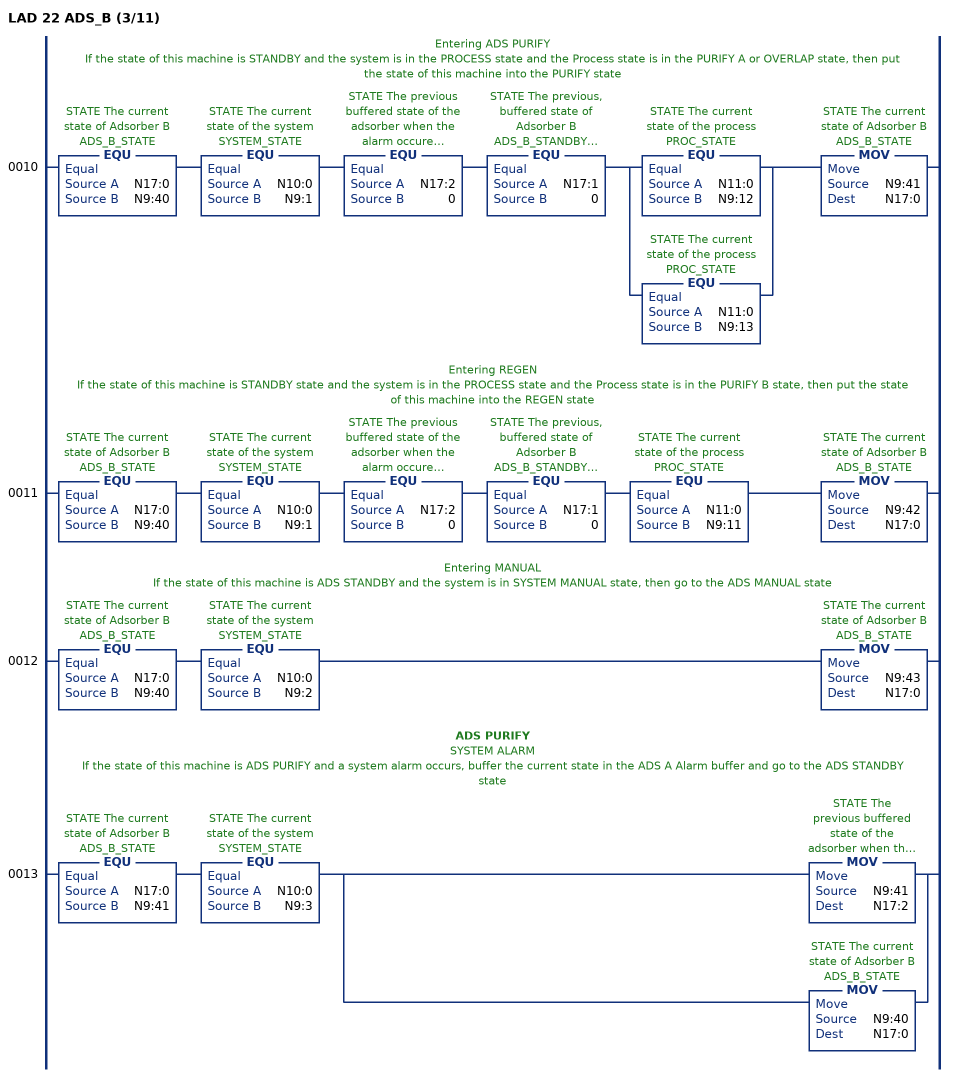
% Rung: 10 %
% Entering ADS PURIFY
% If the state of this machine is STANDBY and the system is in the PROCESS state and the Process state is in the PURIFY A or OVERLAP state, then put the state of this machine into the PURIFY state %
SOR EQU N17:0 N9:40 EQU N10:0 N9:1 EQU N17:2 0 EQU N17:1 0 BST EQU N11:0 N9:12 NXB EQU N11:0 N9:13 BND MOV N9:41 N17:0 EOR
%   N17:0  ADS_B_STATE  "STATE The current state of Adsorber B" %
%   N9:40  ADS_STANDBY  "STATE ADS Standby" %
%   N10:0  SYSTEM_STATE  "STATE The current state of the system" %
%   N9:1  SYSTEM_PROCESS  "STATE System Process" %
%   N17:2  ADS_B_SYS_ALARM_BUFR  "STATE The previous buffered state of the adsorber when the alarm occured" %
%   N17:1  ADS_B_STANDBY_BUFFER  "STATE The previous, buffered state of Adsorber B" %
%   N11:0  PROC_STATE  "STATE The current state of the process" %
%   N9:12  PROC_PURIFY_B  "STATE Process Purify B" %
%   N9:13  PROC_OVERLAP  "STATE Process Purify Overlap" %
%   N9:41  ADS_PURIFY  "STATE ADS Purify" %
% Rung: 11 %
% Entering REGEN
% If the state of this machine is STANDBY state and the system is in the PROCESS state and the Process state is in the PURIFY B state, then put the state of this machine into the REGEN state %
SOR EQU N17:0 N9:40 EQU N10:0 N9:1 EQU N17:2 0 EQU N17:1 0 EQU N11:0 N9:11 MOV N9:42 N17:0 EOR
%   N17:0  ADS_B_STATE  "STATE The current state of Adsorber B" %
%   N9:40  ADS_STANDBY  "STATE ADS Standby" %
%   N10:0  SYSTEM_STATE  "STATE The current state of the system" %
%   N9:1  SYSTEM_PROCESS  "STATE System Process" %
%   N17:2  ADS_B_SYS_ALARM_BUFR  "STATE The previous buffered state of the adsorber when the alarm occured" %
%   N17:1  ADS_B_STANDBY_BUFFER  "STATE The previous, buffered state of Adsorber B" %
%   N11:0  PROC_STATE  "STATE The current state of the process" %
%   N9:11  PROC_PURIFY_A  "STATE Process Purify A" %
%   N9:42  ADS_REGEN  "STATE ADS Regen" %
% Rung: 12 %
% Entering MANUAL
% If the state of this machine is ADS STANDBY and the system is in SYSTEM MANUAL state, then go to the ADS MANUAL state %
SOR EQU N17:0 N9:40 EQU N10:0 N9:2 MOV N9:43 N17:0 EOR
%   N17:0  ADS_B_STATE  "STATE The current state of Adsorber B" %
%   N9:40  ADS_STANDBY  "STATE ADS Standby" %
%   N10:0  SYSTEM_STATE  "STATE The current state of the system" %
%   N9:2  SYSTEM_MANUAL  "STATE System Manual" %
%   N9:43  ADS_MANUAL  "STATE ADS Manual" %
% Rung: 13 %
% TITLE: ADS PURIFY %
% SYSTEM ALARM
% If the state of this machine is ADS PURIFY and a system alarm occurs, buffer the current state in the ADS A Alarm buffer and go to the ADS STANDBY state %
SOR EQU N17:0 N9:41 EQU N10:0 N9:3 BST MOV N9:41 N17:2 NXB MOV N9:40 N17:0 BND EOR
%   N17:0  ADS_B_STATE  "STATE The current state of Adsorber B" %
%   N9:41  ADS_PURIFY  "STATE ADS Purify" %
%   N10:0  SYSTEM_STATE  "STATE The current state of the system" %
%   N9:3  SYSTEM_ALARM  "STATE System Alarm" %
%   N17:2  ADS_B_SYS_ALARM_BUFR  "STATE The previous buffered state of the adsorber when the alarm occured" %
%   N9:40  ADS_STANDBY  "STATE ADS Standby" %

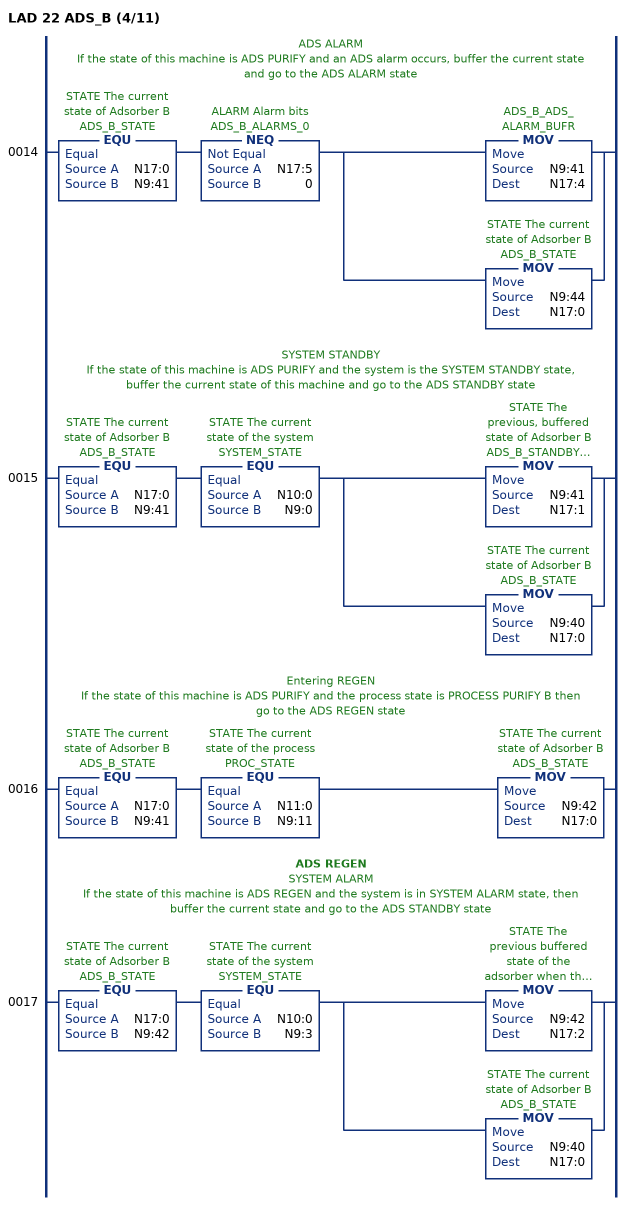
% Rung: 14 %
% ADS ALARM
% If the state of this machine is ADS PURIFY and an ADS alarm occurs, buffer the current state and go to the ADS ALARM state %
SOR EQU N17:0 N9:41 NEQ N17:5 0 BST MOV N9:41 N17:4 NXB MOV N9:44 N17:0 BND EOR
%   N17:0  ADS_B_STATE  "STATE The current state of Adsorber B" %
%   N9:41  ADS_PURIFY  "STATE ADS Purify" %
%   N17:5  ADS_B_ALARMS_0  "ALARM Alarm bits" %
%   N17:4  ADS_B_ADS_ALARM_BUFR %
%   N9:44  ADS_ALARM  "STATE ADS Alarm" %
% Rung: 15 %
% SYSTEM STANDBY
% If the state of this machine is ADS PURIFY and the system is the SYSTEM STANDBY state, buffer the current state of this machine and go to the ADS STANDBY state %
SOR EQU N17:0 N9:41 EQU N10:0 N9:0 BST MOV N9:41 N17:1 NXB MOV N9:40 N17:0 BND EOR
%   N17:0  ADS_B_STATE  "STATE The current state of Adsorber B" %
%   N9:41  ADS_PURIFY  "STATE ADS Purify" %
%   N10:0  SYSTEM_STATE  "STATE The current state of the system" %
%   N9:0  SYSTEM_STANDBY  "STATE System Standby" %
%   N17:1  ADS_B_STANDBY_BUFFER  "STATE The previous, buffered state of Adsorber B" %
%   N9:40  ADS_STANDBY  "STATE ADS Standby" %
% Rung: 16 %
% Entering REGEN
% If the state of this machine is ADS PURIFY and the process state is PROCESS PURIFY B then go to the ADS REGEN state %
SOR EQU N17:0 N9:41 EQU N11:0 N9:11 MOV N9:42 N17:0 EOR
%   N17:0  ADS_B_STATE  "STATE The current state of Adsorber B" %
%   N9:41  ADS_PURIFY  "STATE ADS Purify" %
%   N11:0  PROC_STATE  "STATE The current state of the process" %
%   N9:11  PROC_PURIFY_A  "STATE Process Purify A" %
%   N9:42  ADS_REGEN  "STATE ADS Regen" %
% Rung: 17 %
% TITLE: ADS REGEN %
% SYSTEM ALARM
% If the state of this machine is ADS REGEN and the system is in SYSTEM ALARM state, then buffer the current state and go to the ADS STANDBY state %
SOR EQU N17:0 N9:42 EQU N10:0 N9:3 BST MOV N9:42 N17:2 NXB MOV N9:40 N17:0 BND EOR
%   N17:0  ADS_B_STATE  "STATE The current state of Adsorber B" %
%   N9:42  ADS_REGEN  "STATE ADS Regen" %
%   N10:0  SYSTEM_STATE  "STATE The current state of the system" %
%   N9:3  SYSTEM_ALARM  "STATE System Alarm" %
%   N17:2  ADS_B_SYS_ALARM_BUFR  "STATE The previous buffered state of the adsorber when the alarm occured" %
%   N9:40  ADS_STANDBY  "STATE ADS Standby" %

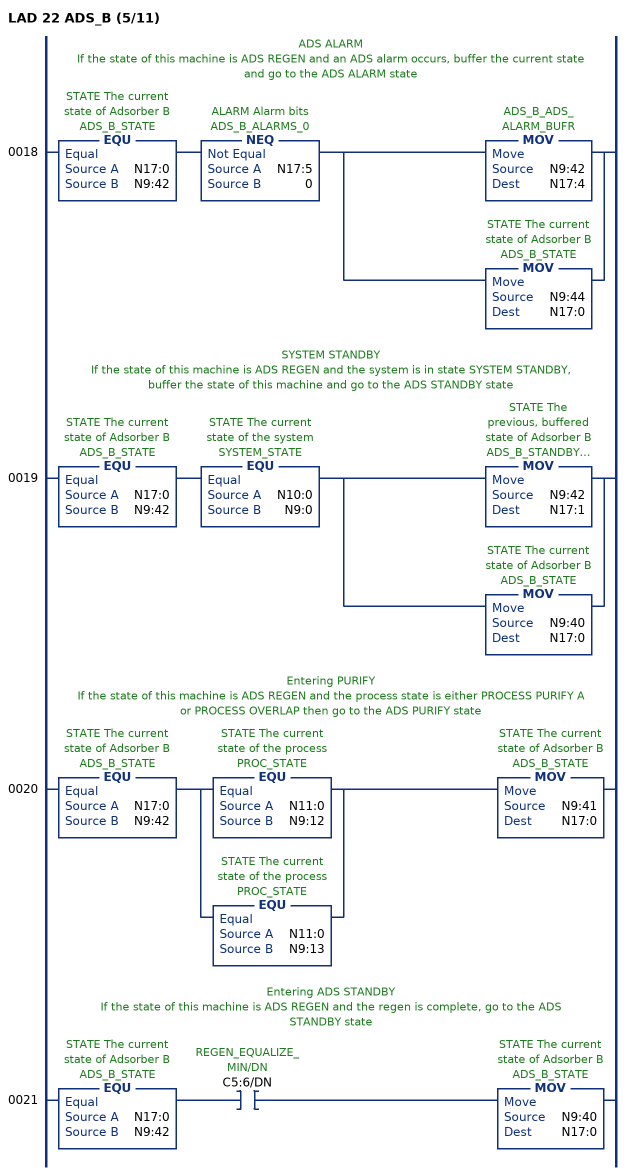
% Rung: 18 %
% ADS ALARM
% If the state of this machine is ADS REGEN and an ADS alarm occurs, buffer the current state and go to the ADS ALARM state %
SOR EQU N17:0 N9:42 NEQ N17:5 0 BST MOV N9:42 N17:4 NXB MOV N9:44 N17:0 BND EOR
%   N17:0  ADS_B_STATE  "STATE The current state of Adsorber B" %
%   N9:42  ADS_REGEN  "STATE ADS Regen" %
%   N17:5  ADS_B_ALARMS_0  "ALARM Alarm bits" %
%   N17:4  ADS_B_ADS_ALARM_BUFR %
%   N9:44  ADS_ALARM  "STATE ADS Alarm" %
% Rung: 19 %
% SYSTEM STANDBY
% If the state of this machine is ADS REGEN and the system is in state SYSTEM STANDBY, buffer the state of this machine and go to the ADS STANDBY state %
SOR EQU N17:0 N9:42 EQU N10:0 N9:0 BST MOV N9:42 N17:1 NXB MOV N9:40 N17:0 BND EOR
%   N17:0  ADS_B_STATE  "STATE The current state of Adsorber B" %
%   N9:42  ADS_REGEN  "STATE ADS Regen" %
%   N10:0  SYSTEM_STATE  "STATE The current state of the system" %
%   N9:0  SYSTEM_STANDBY  "STATE System Standby" %
%   N17:1  ADS_B_STANDBY_BUFFER  "STATE The previous, buffered state of Adsorber B" %
%   N9:40  ADS_STANDBY  "STATE ADS Standby" %
% Rung: 20 %
% Entering PURIFY
% If the state of this machine is ADS REGEN and the process state is either PROCESS PURIFY A or PROCESS OVERLAP then go to the ADS PURIFY state %
SOR EQU N17:0 N9:42 BST EQU N11:0 N9:12 NXB EQU N11:0 N9:13 BND MOV N9:41 N17:0 EOR
%   N17:0  ADS_B_STATE  "STATE The current state of Adsorber B" %
%   N9:42  ADS_REGEN  "STATE ADS Regen" %
%   N11:0  PROC_STATE  "STATE The current state of the process" %
%   N9:12  PROC_PURIFY_B  "STATE Process Purify B" %
%   N9:13  PROC_OVERLAP  "STATE Process Purify Overlap" %
%   N9:41  ADS_PURIFY  "STATE ADS Purify" %
% Rung: 21 %
% Entering ADS STANDBY
% If the state of this machine is ADS REGEN and the regen is complete, go to the ADS STANDBY state %
SOR EQU N17:0 N9:42 XIC C5:6/DN MOV N9:40 N17:0 EOR
%   N17:0  ADS_B_STATE  "STATE The current state of Adsorber B" %
%   N9:42  ADS_REGEN  "STATE ADS Regen" %
%   C5:6  REGEN_EQUALIZE_MIN %
%   N9:40  ADS_STANDBY  "STATE ADS Standby" %

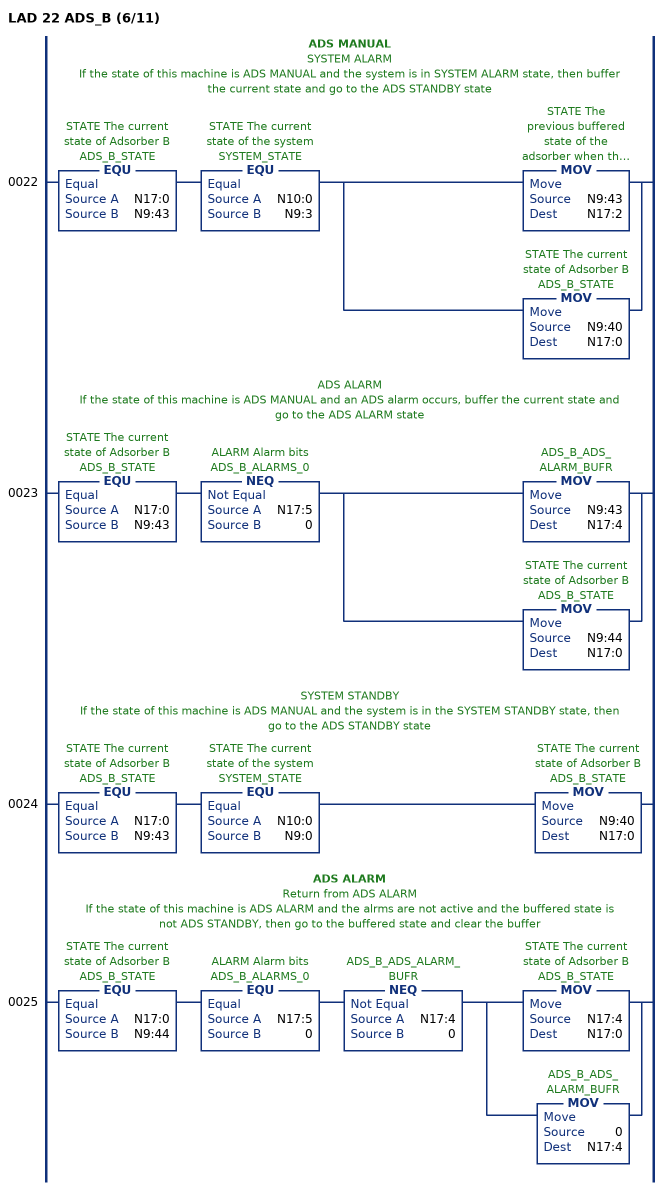
% Rung: 22 %
% TITLE: ADS MANUAL %
% SYSTEM ALARM
% If the state of this machine is ADS MANUAL and the system is in SYSTEM ALARM state, then buffer the current state and go to the ADS STANDBY state %
SOR EQU N17:0 N9:43 EQU N10:0 N9:3 BST MOV N9:43 N17:2 NXB MOV N9:40 N17:0 BND EOR
%   N17:0  ADS_B_STATE  "STATE The current state of Adsorber B" %
%   N9:43  ADS_MANUAL  "STATE ADS Manual" %
%   N10:0  SYSTEM_STATE  "STATE The current state of the system" %
%   N9:3  SYSTEM_ALARM  "STATE System Alarm" %
%   N17:2  ADS_B_SYS_ALARM_BUFR  "STATE The previous buffered state of the adsorber when the alarm occured" %
%   N9:40  ADS_STANDBY  "STATE ADS Standby" %
% Rung: 23 %
% ADS ALARM
% If the state of this machine is ADS MANUAL and an ADS alarm occurs, buffer the current state and go to the ADS ALARM state %
SOR EQU N17:0 N9:43 NEQ N17:5 0 BST MOV N9:43 N17:4 NXB MOV N9:44 N17:0 BND EOR
%   N17:0  ADS_B_STATE  "STATE The current state of Adsorber B" %
%   N9:43  ADS_MANUAL  "STATE ADS Manual" %
%   N17:5  ADS_B_ALARMS_0  "ALARM Alarm bits" %
%   N17:4  ADS_B_ADS_ALARM_BUFR %
%   N9:44  ADS_ALARM  "STATE ADS Alarm" %
% Rung: 24 %
% SYSTEM STANDBY
% If the state of this machine is ADS MANUAL and the system is in the SYSTEM STANDBY state, then go to the ADS STANDBY state %
SOR EQU N17:0 N9:43 EQU N10:0 N9:0 MOV N9:40 N17:0 EOR
%   N17:0  ADS_B_STATE  "STATE The current state of Adsorber B" %
%   N9:43  ADS_MANUAL  "STATE ADS Manual" %
%   N10:0  SYSTEM_STATE  "STATE The current state of the system" %
%   N9:0  SYSTEM_STANDBY  "STATE System Standby" %
%   N9:40  ADS_STANDBY  "STATE ADS Standby" %
% Rung: 25 %
% TITLE: ADS ALARM %
% Return from ADS ALARM
% If the state of this machine is ADS ALARM and the alrms are not active and the buffered state is not ADS STANDBY, then go to the buffered state and clear the buffer %
SOR EQU N17:0 N9:44 EQU N17:5 0 NEQ N17:4 0 BST MOV N17:4 N17:0 NXB MOV 0 N17:4 BND EOR
%   N17:0  ADS_B_STATE  "STATE The current state of Adsorber B" %
%   N9:44  ADS_ALARM  "STATE ADS Alarm" %
%   N17:5  ADS_B_ALARMS_0  "ALARM Alarm bits" %
%   N17:4  ADS_B_ADS_ALARM_BUFR %

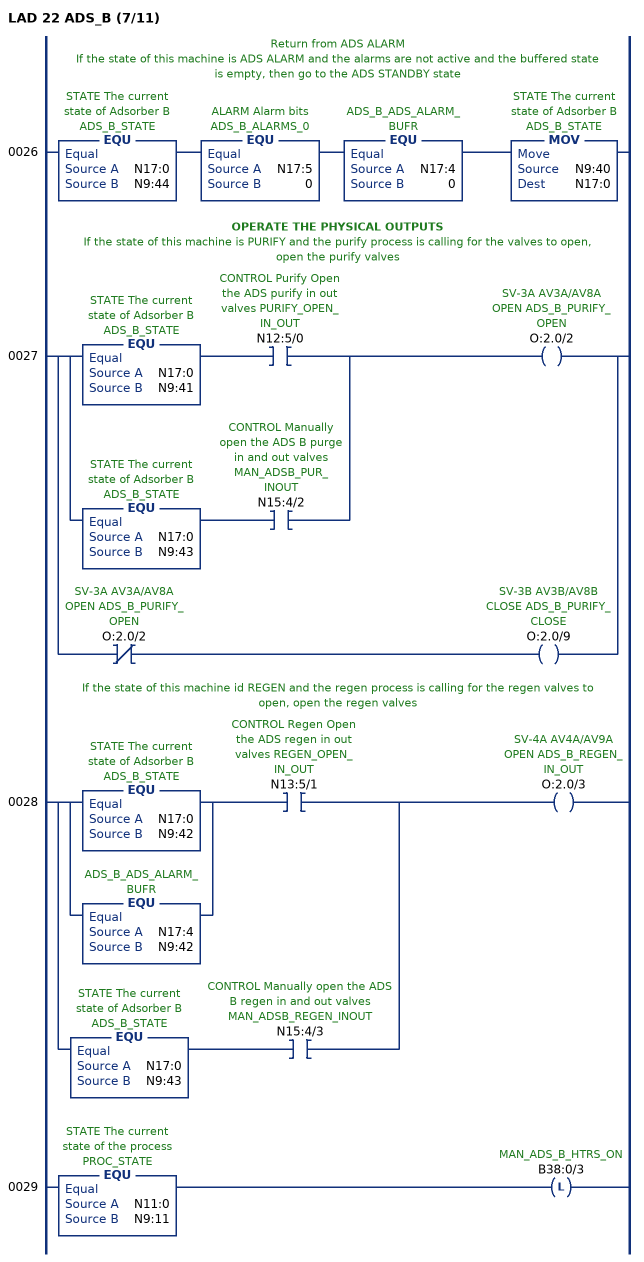
% Rung: 26 %
% Return from ADS ALARM
% If the state of this machine is ADS ALARM and the alarms are not active and the buffered state is empty, then go to the ADS STANDBY state %
SOR EQU N17:0 N9:44 EQU N17:5 0 EQU N17:4 0 MOV N9:40 N17:0 EOR
%   N17:0  ADS_B_STATE  "STATE The current state of Adsorber B" %
%   N9:44  ADS_ALARM  "STATE ADS Alarm" %
%   N17:5  ADS_B_ALARMS_0  "ALARM Alarm bits" %
%   N17:4  ADS_B_ADS_ALARM_BUFR %
%   N9:40  ADS_STANDBY  "STATE ADS Standby" %
% Rung: 27 %
% TITLE: OPERATE THE PHYSICAL OUTPUTS %
% If the state of this machine is PURIFY and the purify process is calling for the valves to open, open the purify valves %
SOR BST BST EQU N17:0 N9:41 XIC N12:5/0 NXB EQU N17:0 N9:43 XIC N15:4/2 BND OTE O:2.0/2 NXB XIO O:2.0/2 OTE O:2.0/9 BND EOR
%   N17:0  ADS_B_STATE  "STATE The current state of Adsorber B" %
%   N9:41  ADS_PURIFY  "STATE ADS Purify" %
%   N12:5/0  PURIFY_OPEN_IN_OUT  "CONTROL Purify Open the ADS purify in out valves" %
%   N9:43  ADS_MANUAL  "STATE ADS Manual" %
%   N15:4/2  MAN_ADSB_PUR_INOUT  "CONTROL Manually open the ADS B purge in and out valves" %
%   O:2.0/2  ADS_B_PURIFY_OPEN  "SV-3A AV3A/AV8A OPEN" %
%   O:2.0/9  ADS_B_PURIFY_CLOSE  "SV-3B AV3B/AV8B CLOSE" %
% Rung: 28 %
% If the state of this machine id REGEN and the regen process is calling for the regen valves to open, open the regen valves %
SOR BST BST EQU N17:0 N9:42 NXB EQU N17:4 N9:42 BND XIC N13:5/1 NXB EQU N17:0 N9:43 XIC N15:4/3 BND OTE O:2.0/3 EOR
%   N17:0  ADS_B_STATE  "STATE The current state of Adsorber B" %
%   N9:42  ADS_REGEN  "STATE ADS Regen" %
%   N17:4  ADS_B_ADS_ALARM_BUFR %
%   N13:5/1  REGEN_OPEN_IN_OUT  "CONTROL Regen Open the ADS regen in out valves" %
%   N9:43  ADS_MANUAL  "STATE ADS Manual" %
%   N15:4/3  MAN_ADSB_REGEN_INOUT  "CONTROL Manually open the ADS B regen in and out valves" %
%   O:2.0/3  ADS_B_REGEN_IN_OUT  "SV-4A AV4A/AV9A OPEN" %
% Rung: 29 %
SOR EQU N11:0 N9:11 OTL B38:0/3 EOR
%   N11:0  PROC_STATE  "STATE The current state of the process" %
%   N9:11  PROC_PURIFY_A  "STATE Process Purify A" %
%   B38:0/3  MAN_ADS_B_HTRS_ON %

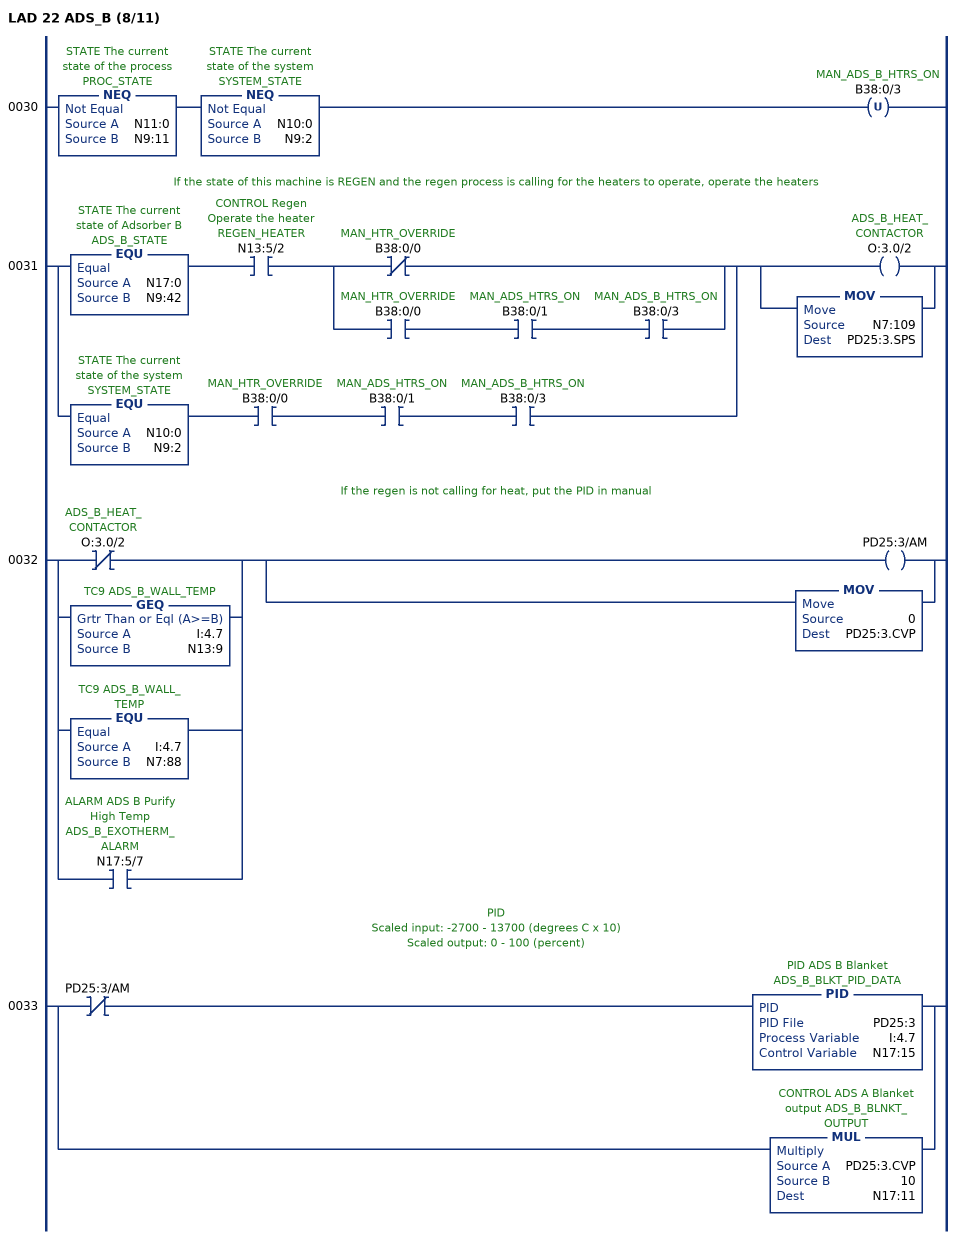
% Rung: 30 %
SOR NEQ N11:0 N9:11 NEQ N10:0 N9:2 OTU B38:0/3 EOR
%   N11:0  PROC_STATE  "STATE The current state of the process" %
%   N9:11  PROC_PURIFY_A  "STATE Process Purify A" %
%   N10:0  SYSTEM_STATE  "STATE The current state of the system" %
%   N9:2  SYSTEM_MANUAL  "STATE System Manual" %
%   B38:0/3  MAN_ADS_B_HTRS_ON %
% Rung: 31 %
% If the state of this machine is REGEN and the regen process is calling for the heaters to operate, operate the heaters %
SOR BST EQU N17:0 N9:42 XIC N13:5/2 BST XIO B38:0/0 NXB XIC B38:0/0 XIC B38:0/1 XIC B38:0/3 BND NXB EQU N10:0 N9:2 XIC B38:0/0 XIC B38:0/1 XIC B38:0/3 BND BST OTE O:3.0/2 NXB MOV N7:109 PD25:3.SPS BND EOR
%   N17:0  ADS_B_STATE  "STATE The current state of Adsorber B" %
%   N9:42  ADS_REGEN  "STATE ADS Regen" %
%   N13:5/2  REGEN_HEATER  "CONTROL Regen Operate the heater" %
%   B38:0/0  MAN_HTR_OVERRIDE %
%   B38:0/1  MAN_ADS_HTRS_ON %
%   B38:0/3  MAN_ADS_B_HTRS_ON %
%   N10:0  SYSTEM_STATE  "STATE The current state of the system" %
%   N9:2  SYSTEM_MANUAL  "STATE System Manual" %
%   O:3.0/2  ADS_B_HEAT_CONTACTOR %
%   N7:109  BLANKET_SP  "CONTROL Blanket PID Setpoint" %
% Rung: 32 %
% If the regen is not calling for heat, put the PID in manual %
SOR BST XIO O:3.0/2 NXB GEQ I:4.7 N13:9 NXB EQU I:4.7 N7:88 NXB XIC N17:5/7 BND BST OTE PD25:3/AM NXB MOV 0 PD25:3.CVP BND EOR
%   O:3.0/2  ADS_B_HEAT_CONTACTOR %
%   I:4.7  ADS_B_WALL_TEMP  "TC9" %
%   N13:9  BLANKET_LIMIT %
%   N7:88  TC_OPEN_SP  "CONFIG The value read by an open TC input" %
%   N17:5/7  ADS_B_EXOTHERM_ALARM  "ALARM ADS B Purify High Temp" %
% Rung: 33 %
% PID
% Scaled input: -2700 - 13700 (degrees C x 10)
% Scaled output: 0 - 100 (percent) %
SOR BST XIO PD25:3/AM PID PD25:3 I:4.7 N17:15 NXB MUL PD25:3.CVP 10 N17:11 BND EOR
%   PD25:3  ADS_B_BLKT_PID_DATA  "PID ADS B Blanket" %
%   I:4.7  ADS_B_WALL_TEMP  "TC9" %
%   N17:15  ADS_B_BLKT_OUTPT_RAW  "CONTROL ADS B Blanket PID Output Raw" %
%   N17:11  ADS_B_BLNKT_OUTPUT  "CONTROL ADS A Blanket output" %

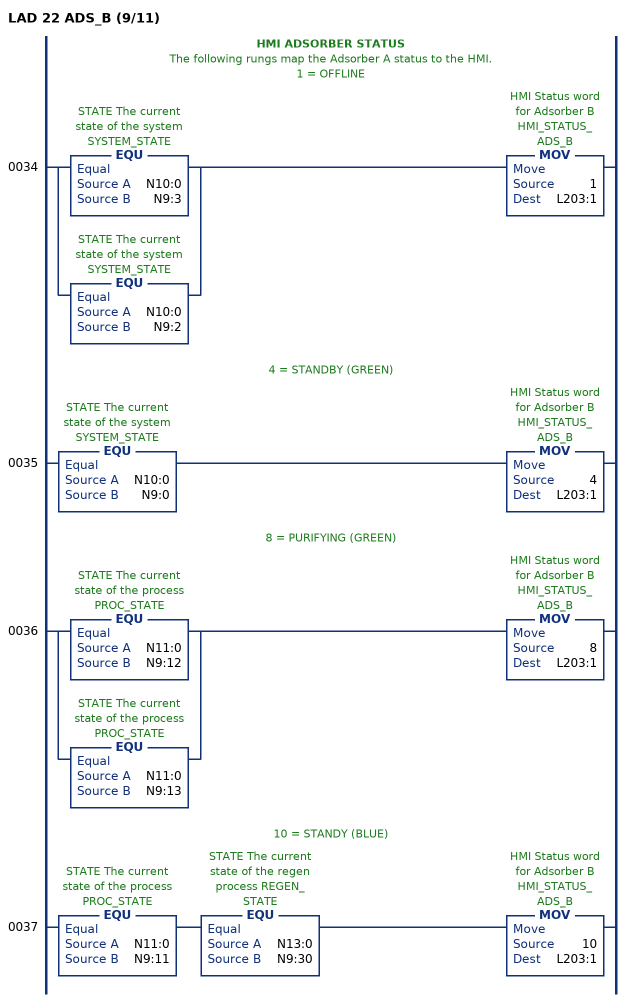
% Rung: 34 %
% TITLE: HMI ADSORBER STATUS %
% The following rungs map the Adsorber A status to the HMI.
% 1 = OFFLINE %
SOR BST EQU N10:0 N9:3 NXB EQU N10:0 N9:2 BND MOV 1 L203:1 EOR
%   N10:0  SYSTEM_STATE  "STATE The current state of the system" %
%   N9:3  SYSTEM_ALARM  "STATE System Alarm" %
%   N9:2  SYSTEM_MANUAL  "STATE System Manual" %
%   L203:1  HMI_STATUS_ADS_B  "HMI Status word for Adsorber B" %
% Rung: 35 %
% 4 = STANDBY (GREEN) %
SOR EQU N10:0 N9:0 MOV 4 L203:1 EOR
%   N10:0  SYSTEM_STATE  "STATE The current state of the system" %
%   N9:0  SYSTEM_STANDBY  "STATE System Standby" %
%   L203:1  HMI_STATUS_ADS_B  "HMI Status word for Adsorber B" %
% Rung: 36 %
% 8 = PURIFYING (GREEN) %
SOR BST EQU N11:0 N9:12 NXB EQU N11:0 N9:13 BND MOV 8 L203:1 EOR
%   N11:0  PROC_STATE  "STATE The current state of the process" %
%   N9:12  PROC_PURIFY_B  "STATE Process Purify B" %
%   N9:13  PROC_OVERLAP  "STATE Process Purify Overlap" %
%   L203:1  HMI_STATUS_ADS_B  "HMI Status word for Adsorber B" %
% Rung: 37 %
% 10 = STANDY (BLUE) %
SOR EQU N11:0 N9:11 EQU N13:0 N9:30 MOV 10 L203:1 EOR
%   N11:0  PROC_STATE  "STATE The current state of the process" %
%   N9:11  PROC_PURIFY_A  "STATE Process Purify A" %
%   N13:0  REGEN_STATE  "STATE The current state of the regen process" %
%   N9:30  REGEN_STANDBY  "STATE Regen Standby" %
%   L203:1  HMI_STATUS_ADS_B  "HMI Status word for Adsorber B" %

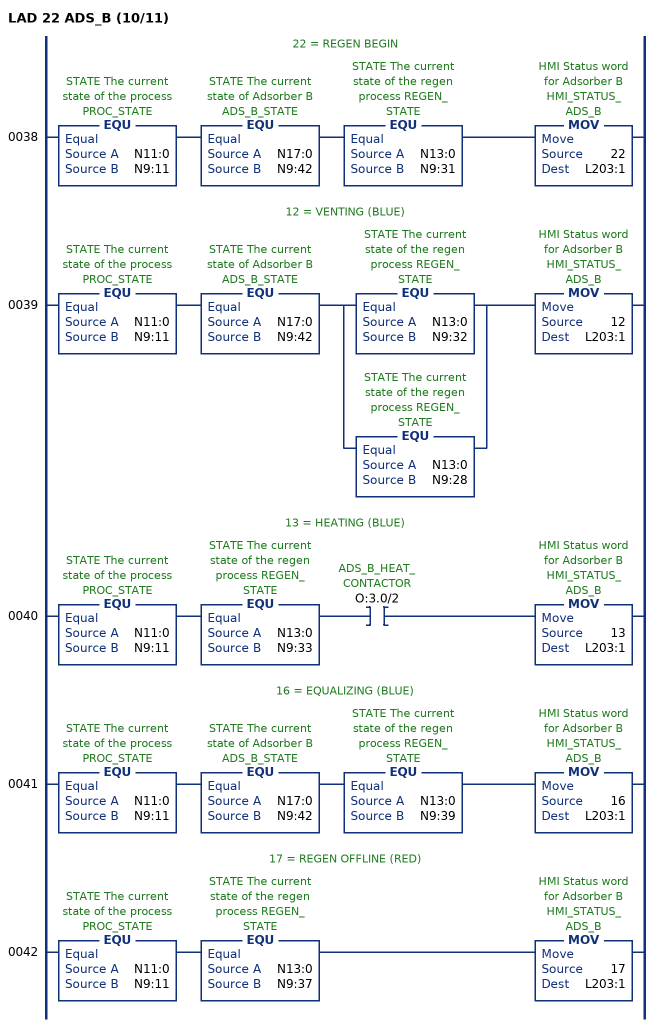
% Rung: 38 %
% 22 = REGEN BEGIN %
SOR EQU N11:0 N9:11 EQU N17:0 N9:42 EQU N13:0 N9:31 MOV 22 L203:1 EOR
%   N11:0  PROC_STATE  "STATE The current state of the process" %
%   N9:11  PROC_PURIFY_A  "STATE Process Purify A" %
%   N17:0  ADS_B_STATE  "STATE The current state of Adsorber B" %
%   N9:42  ADS_REGEN  "STATE ADS Regen" %
%   N13:0  REGEN_STATE  "STATE The current state of the regen process" %
%   N9:31  REGEN_DELAY  "STATE Regen Delay" %
%   L203:1  HMI_STATUS_ADS_B  "HMI Status word for Adsorber B" %
% Rung: 39 %
% 12 = VENTING (BLUE) %
SOR EQU N11:0 N9:11 EQU N17:0 N9:42 BST EQU N13:0 N9:32 NXB EQU N13:0 N9:28 BND MOV 12 L203:1 EOR
%   N11:0  PROC_STATE  "STATE The current state of the process" %
%   N9:11  PROC_PURIFY_A  "STATE Process Purify A" %
%   N17:0  ADS_B_STATE  "STATE The current state of Adsorber B" %
%   N9:42  ADS_REGEN  "STATE ADS Regen" %
%   N13:0  REGEN_STATE  "STATE The current state of the regen process" %
%   N9:32  REGEN_VENT  "STATE Regen Vent" %
%   N9:28  REGEN_VENT_2  "STATE Regen Vent 2" %
%   L203:1  HMI_STATUS_ADS_B  "HMI Status word for Adsorber B" %
% Rung: 40 %
% 13 = HEATING (BLUE) %
SOR EQU N11:0 N9:11 EQU N13:0 N9:33 XIC O:3.0/2 MOV 13 L203:1 EOR
%   N11:0  PROC_STATE  "STATE The current state of the process" %
%   N9:11  PROC_PURIFY_A  "STATE Process Purify A" %
%   N13:0  REGEN_STATE  "STATE The current state of the regen process" %
%   N9:33  REGEN_HEAT_BED  "STATE Regen Heat wall" %
%   O:3.0/2  ADS_B_HEAT_CONTACTOR %
%   L203:1  HMI_STATUS_ADS_B  "HMI Status word for Adsorber B" %
% Rung: 41 %
% 16 = EQUALIZING (BLUE) %
SOR EQU N11:0 N9:11 EQU N17:0 N9:42 EQU N13:0 N9:39 MOV 16 L203:1 EOR
%   N11:0  PROC_STATE  "STATE The current state of the process" %
%   N9:11  PROC_PURIFY_A  "STATE Process Purify A" %
%   N17:0  ADS_B_STATE  "STATE The current state of Adsorber B" %
%   N9:42  ADS_REGEN  "STATE ADS Regen" %
%   N13:0  REGEN_STATE  "STATE The current state of the regen process" %
%   N9:39  REGEN_EQUALIZE %
%   L203:1  HMI_STATUS_ADS_B  "HMI Status word for Adsorber B" %
% Rung: 42 %
% 17 = REGEN OFFLINE (RED) %
SOR EQU N11:0 N9:11 EQU N13:0 N9:37 MOV 17 L203:1 EOR
%   N11:0  PROC_STATE  "STATE The current state of the process" %
%   N9:11  PROC_PURIFY_A  "STATE Process Purify A" %
%   N13:0  REGEN_STATE  "STATE The current state of the regen process" %
%   N9:37  REGEN_ALARM  "STATE Regen Alarm" %
%   L203:1  HMI_STATUS_ADS_B  "HMI Status word for Adsorber B" %

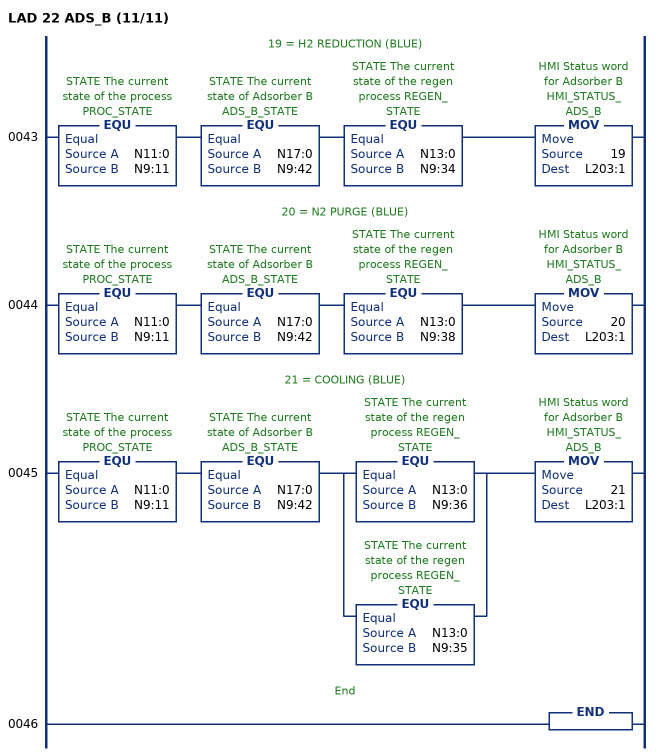
% Rung: 43 %
% 19 = H2 REDUCTION (BLUE) %
SOR EQU N11:0 N9:11 EQU N17:0 N9:42 EQU N13:0 N9:34 MOV 19 L203:1 EOR
%   N11:0  PROC_STATE  "STATE The current state of the process" %
%   N9:11  PROC_PURIFY_A  "STATE Process Purify A" %
%   N17:0  ADS_B_STATE  "STATE The current state of Adsorber B" %
%   N9:42  ADS_REGEN  "STATE ADS Regen" %
%   N13:0  REGEN_STATE  "STATE The current state of the regen process" %
%   N9:34  REGEN_H2_REDUCTION  "STATE Regen Running" %
%   L203:1  HMI_STATUS_ADS_B  "HMI Status word for Adsorber B" %
% Rung: 44 %
% 20 = N2 PURGE (BLUE) %
SOR EQU N11:0 N9:11 EQU N17:0 N9:42 EQU N13:0 N9:38 MOV 20 L203:1 EOR
%   N11:0  PROC_STATE  "STATE The current state of the process" %
%   N9:11  PROC_PURIFY_A  "STATE Process Purify A" %
%   N17:0  ADS_B_STATE  "STATE The current state of Adsorber B" %
%   N9:42  ADS_REGEN  "STATE ADS Regen" %
%   N13:0  REGEN_STATE  "STATE The current state of the regen process" %
%   N9:38  REGEN_PURGE  "STATE Regen Hot Purge" %
%   L203:1  HMI_STATUS_ADS_B  "HMI Status word for Adsorber B" %
% Rung: 45 %
% 21 = COOLING (BLUE) %
SOR EQU N11:0 N9:11 EQU N17:0 N9:42 BST EQU N13:0 N9:36 NXB EQU N13:0 N9:35 BND MOV 21 L203:1 EOR
%   N11:0  PROC_STATE  "STATE The current state of the process" %
%   N9:11  PROC_PURIFY_A  "STATE Process Purify A" %
%   N17:0  ADS_B_STATE  "STATE The current state of Adsorber B" %
%   N9:42  ADS_REGEN  "STATE ADS Regen" %
%   N13:0  REGEN_STATE  "STATE The current state of the regen process" %
%   N9:36  REGEN_COOL  "STATE Regen Cool" %
%   N9:35  REGEN_COOL_WALL  "STATE Regen Cool wall" %
%   L203:1  HMI_STATUS_ADS_B  "HMI Status word for Adsorber B" %
% Rung: 46 %
% End %
SOR END EOR

LADDER 23 "ADS_B_FLT"    % Controls the Adsorber B faults %
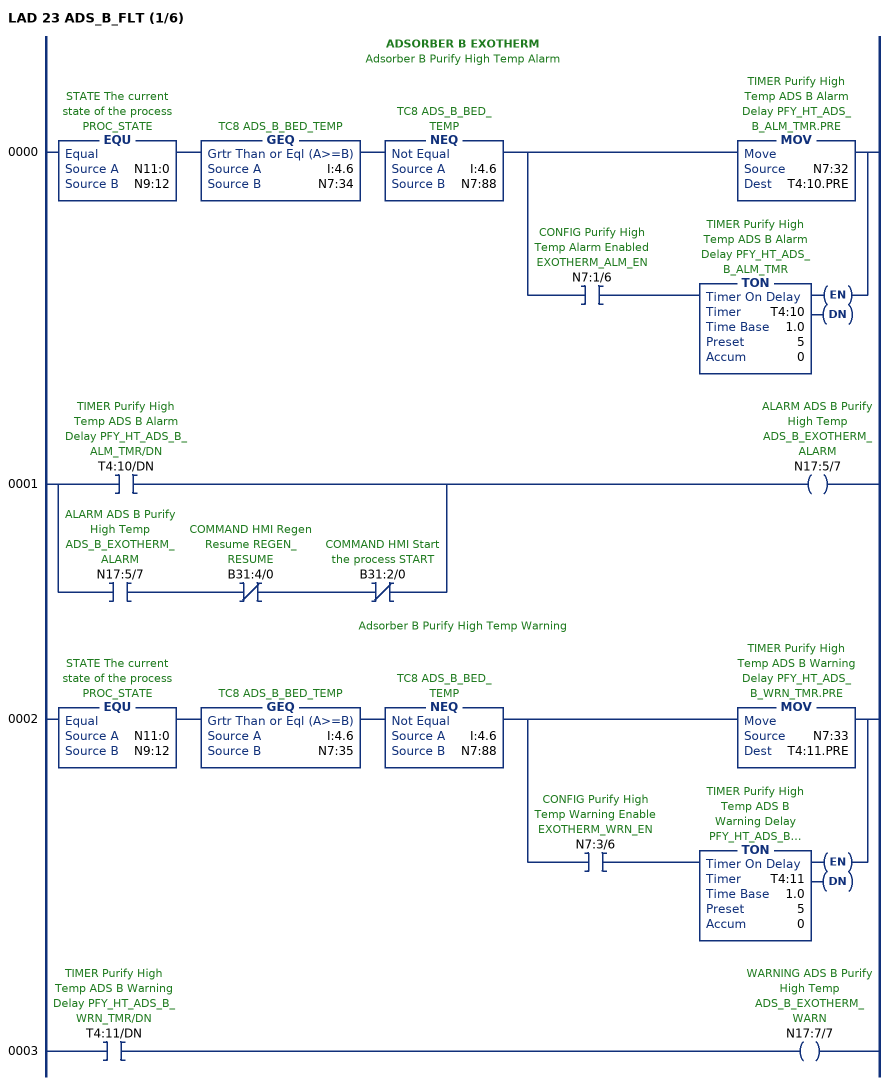
% Rung: 0 %
% TITLE: ADSORBER B EXOTHERM %
% Adsorber B Purify High Temp Alarm %
SOR EQU N11:0 N9:12 GEQ I:4.6 N7:34 NEQ I:4.6 N7:88 BST MOV N7:32 T4:10.PRE NXB XIC N7:1/6 TON T4:10 1.0 5 0 BND EOR
%   N11:0  PROC_STATE  "STATE The current state of the process" %
%   N9:12  PROC_PURIFY_B  "STATE Process Purify B" %
%   I:4.6  ADS_B_BED_TEMP  "TC8" %
%   N7:34  EXOTHERM_ALM_SP  "CONFIG Purify High Temp Alarm Setpoint" %
%   N7:88  TC_OPEN_SP  "CONFIG The value read by an open TC input" %
%   N7:32  EXOTHERM_ALM_DLY  "CONFIG Purify High Temp Alarm Delay" %
%   T4:10  PFY_HT_ADS_B_ALM_TMR  "TIMER Purify High Temp ADS B Alarm Delay" %
%   N7:1/6  EXOTHERM_ALM_EN  "CONFIG Purify High Temp Alarm Enabled" %
% Rung: 1 %
SOR BST XIC T4:10/DN NXB XIC N17:5/7 XIO B31:4/0 XIO B31:2/0 BND OTE N17:5/7 EOR
%   T4:10  PFY_HT_ADS_B_ALM_TMR  "TIMER Purify High Temp ADS B Alarm Delay" %
%   N17:5/7  ADS_B_EXOTHERM_ALARM  "ALARM ADS B Purify High Temp" %
%   B31:4/0  REGEN_RESUME  "COMMAND HMI Regen Resume" %
%   B31:2/0  START  "COMMAND HMI Start the process" %
% Rung: 2 %
% Adsorber B Purify High Temp Warning %
SOR EQU N11:0 N9:12 GEQ I:4.6 N7:35 NEQ I:4.6 N7:88 BST MOV N7:33 T4:11.PRE NXB XIC N7:3/6 TON T4:11 1.0 5 0 BND EOR
%   N11:0  PROC_STATE  "STATE The current state of the process" %
%   N9:12  PROC_PURIFY_B  "STATE Process Purify B" %
%   I:4.6  ADS_B_BED_TEMP  "TC8" %
%   N7:35  EXOTHERM_WRN_SP  "CONFIG Purify High Temp Warning Setpoint" %
%   N7:88  TC_OPEN_SP  "CONFIG The value read by an open TC input" %
%   N7:33  EXOTHERM_WRN_DLY  "CONFIG Purify High Temp Warning Delay" %
%   T4:11  PFY_HT_ADS_B_WRN_TMR  "TIMER Purify High Temp ADS B Warning Delay" %
%   N7:3/6  EXOTHERM_WRN_EN  "CONFIG Purify High Temp Warning Enable" %
% Rung: 3 %
SOR XIC T4:11/DN OTE N17:7/7 EOR
%   T4:11  PFY_HT_ADS_B_WRN_TMR  "TIMER Purify High Temp ADS B Warning Delay" %
%   N17:7/7  ADS_B_EXOTHERM_WARN  "WARNING ADS B Purify High Temp" %

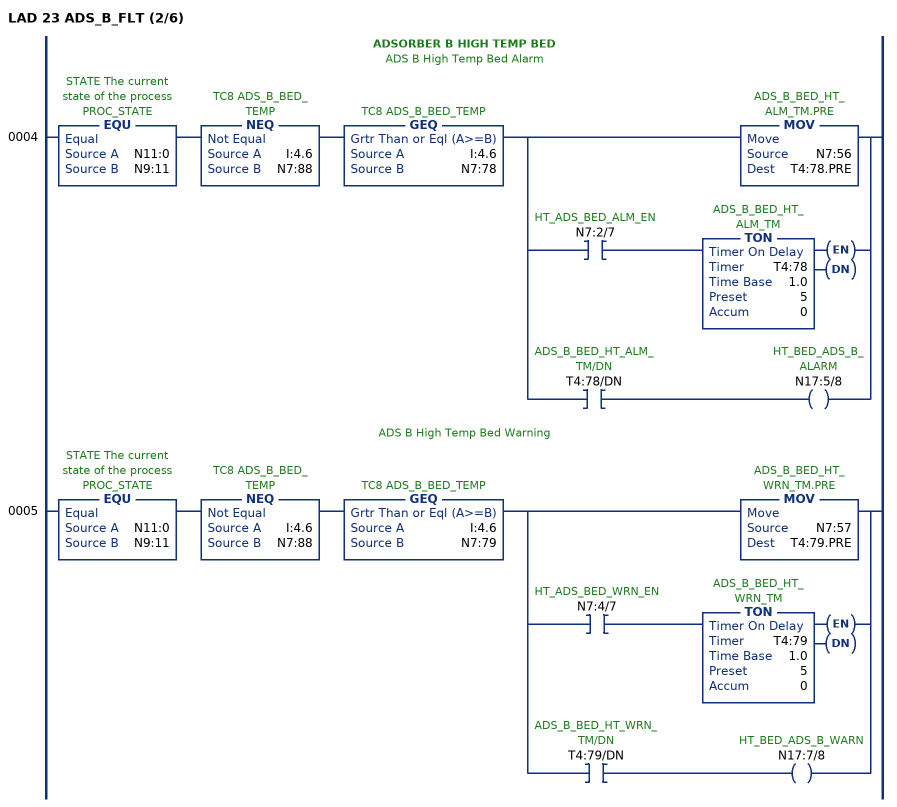
% Rung: 4 %
% TITLE: ADSORBER B HIGH TEMP BED %
% ADS B High Temp Bed Alarm %
SOR EQU N11:0 N9:11 NEQ I:4.6 N7:88 GEQ I:4.6 N7:78 BST MOV N7:56 T4:78.PRE NXB XIC N7:2/7 TON T4:78 1.0 5 0 NXB XIC T4:78/DN OTE N17:5/8 BND EOR
%   N11:0  PROC_STATE  "STATE The current state of the process" %
%   N9:11  PROC_PURIFY_A  "STATE Process Purify A" %
%   I:4.6  ADS_B_BED_TEMP  "TC8" %
%   N7:88  TC_OPEN_SP  "CONFIG The value read by an open TC input" %
%   N7:78  HT_ADS_BED_ALM_SP %
%   N7:56  HT_ADS_BED_ALM_DLY %
%   T4:78  ADS_B_BED_HT_ALM_TM %
%   N7:2/7  HT_ADS_BED_ALM_EN %
%   N17:5/8  HT_BED_ADS_B_ALARM %
% Rung: 5 %
% ADS B High Temp Bed Warning %
SOR EQU N11:0 N9:11 NEQ I:4.6 N7:88 GEQ I:4.6 N7:79 BST MOV N7:57 T4:79.PRE NXB XIC N7:4/7 TON T4:79 1.0 5 0 NXB XIC T4:79/DN OTE N17:7/8 BND EOR
%   N11:0  PROC_STATE  "STATE The current state of the process" %
%   N9:11  PROC_PURIFY_A  "STATE Process Purify A" %
%   I:4.6  ADS_B_BED_TEMP  "TC8" %
%   N7:88  TC_OPEN_SP  "CONFIG The value read by an open TC input" %
%   N7:79  HT_ADS_BED_WRN_SP %
%   N7:57  HT_ADS_BED_WRN_DLY %
%   T4:79  ADS_B_BED_HT_WRN_TM %
%   N7:4/7  HT_ADS_BED_WRN_EN %
%   N17:7/8  HT_BED_ADS_B_WARN %

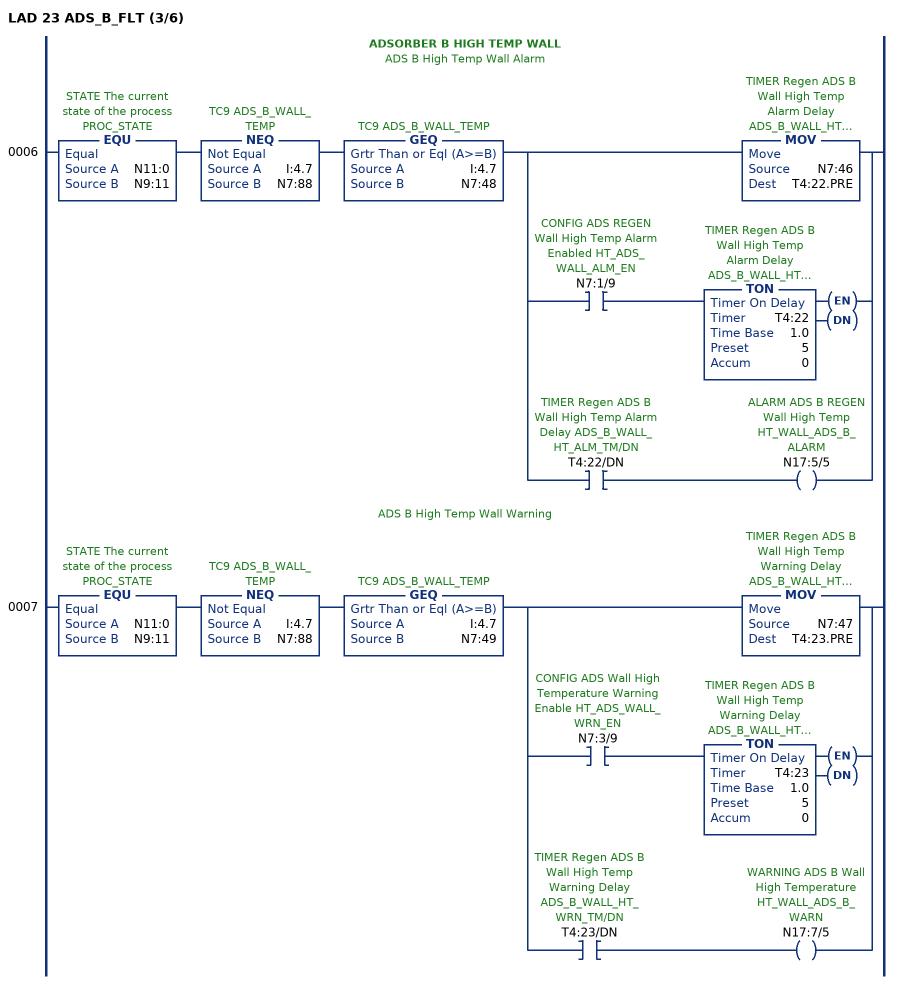
% Rung: 6 %
% TITLE: ADSORBER B HIGH TEMP WALL %
% ADS B High Temp Wall Alarm %
SOR EQU N11:0 N9:11 NEQ I:4.7 N7:88 GEQ I:4.7 N7:48 BST MOV N7:46 T4:22.PRE NXB XIC N7:1/9 TON T4:22 1.0 5 0 NXB XIC T4:22/DN OTE N17:5/5 BND EOR
%   N11:0  PROC_STATE  "STATE The current state of the process" %
%   N9:11  PROC_PURIFY_A  "STATE Process Purify A" %
%   I:4.7  ADS_B_WALL_TEMP  "TC9" %
%   N7:88  TC_OPEN_SP  "CONFIG The value read by an open TC input" %
%   N7:48  HT_ADS_WALL_ALM_SP  "CONFIG ADS Wall Regen High Temp Alarm" %
%   N7:46  HT_ADS_WALL_ALM_DLY  "CONFIG ADS Wall High Temperature Alarm Delay" %
%   T4:22  ADS_B_WALL_HT_ALM_TM  "TIMER Regen ADS B Wall High Temp Alarm Delay" %
%   N7:1/9  HT_ADS_WALL_ALM_EN  "CONFIG ADS REGEN Wall High Temp Alarm Enabled" %
%   N17:5/5  HT_WALL_ADS_B_ALARM  "ALARM ADS B REGEN Wall High Temp" %
% Rung: 7 %
% ADS B High Temp Wall Warning %
SOR EQU N11:0 N9:11 NEQ I:4.7 N7:88 GEQ I:4.7 N7:49 BST MOV N7:47 T4:23.PRE NXB XIC N7:3/9 TON T4:23 1.0 5 0 NXB XIC T4:23/DN OTE N17:7/5 BND EOR
%   N11:0  PROC_STATE  "STATE The current state of the process" %
%   N9:11  PROC_PURIFY_A  "STATE Process Purify A" %
%   I:4.7  ADS_B_WALL_TEMP  "TC9" %
%   N7:88  TC_OPEN_SP  "CONFIG The value read by an open TC input" %
%   N7:49  HT_ADS_WALL_WRN_SP  "CONFIG ADS Wall Regen High Temp Alarm" %
%   N7:47  HT_ADS_WALL_WRN_DLY  "CONFIG ADS Wall High Temperature Warning Delay" %
%   T4:23  ADS_B_WALL_HT_WRN_TM  "TIMER Regen ADS B Wall High Temp Warning Delay" %
%   N7:3/9  HT_ADS_WALL_WRN_EN  "CONFIG ADS Wall High Temperature Warning Enable" %
%   N17:7/5  HT_WALL_ADS_B_WARN  "WARNING ADS B Wall High Temperature" %

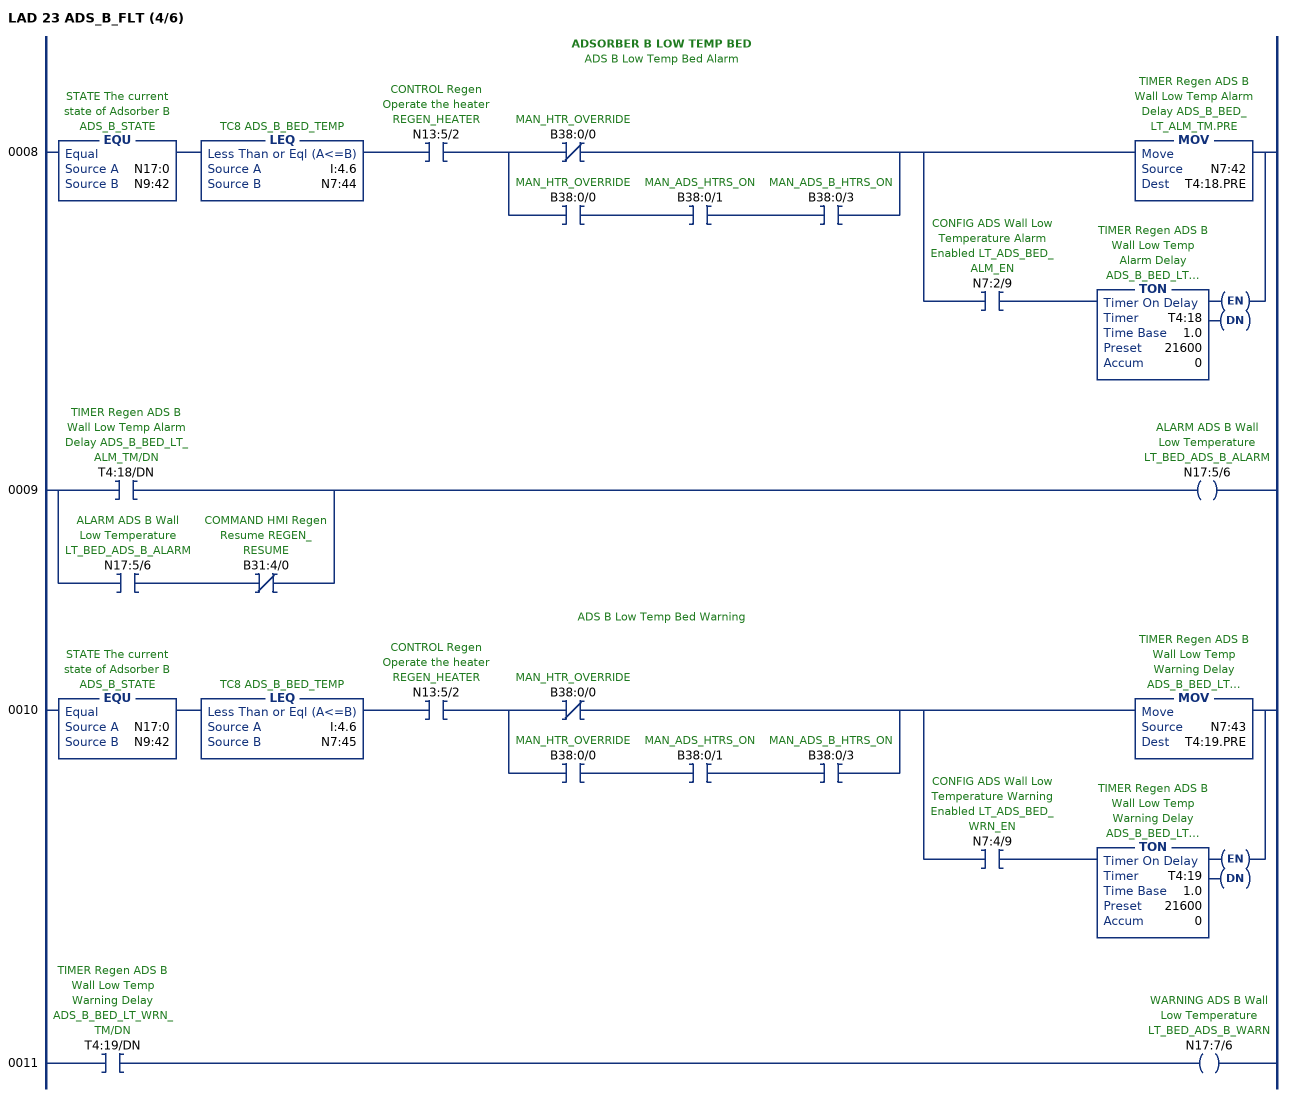
% Rung: 8 %
% TITLE: ADSORBER B LOW TEMP BED %
% ADS B Low Temp Bed Alarm %
SOR EQU N17:0 N9:42 LEQ I:4.6 N7:44 XIC N13:5/2 BST XIO B38:0/0 NXB XIC B38:0/0 XIC B38:0/1 XIC B38:0/3 BND BST MOV N7:42 T4:18.PRE NXB XIC N7:2/9 TON T4:18 1.0 21600 0 BND EOR
%   N17:0  ADS_B_STATE  "STATE The current state of Adsorber B" %
%   N9:42  ADS_REGEN  "STATE ADS Regen" %
%   I:4.6  ADS_B_BED_TEMP  "TC8" %
%   N7:44  LT_ADS_BED_ALM_SP  "CONFIG ADS Wall Regen Heat Low Temperature Alarm Setpoint" %
%   N13:5/2  REGEN_HEATER  "CONTROL Regen Operate the heater" %
%   B38:0/0  MAN_HTR_OVERRIDE %
%   B38:0/1  MAN_ADS_HTRS_ON %
%   B38:0/3  MAN_ADS_B_HTRS_ON %
%   N7:42  LT_ADS_BED_ALM_DLY  "CONFIG ADS Wall Regen heat Low Temperature Alarm Delay" %
%   T4:18  ADS_B_BED_LT_ALM_TM  "TIMER Regen ADS B Wall Low Temp Alarm Delay" %
%   N7:2/9  LT_ADS_BED_ALM_EN  "CONFIG ADS Wall Low Temperature Alarm Enabled" %
% Rung: 9 %
SOR BST XIC T4:18/DN NXB XIC N17:5/6 XIO B31:4/0 BND OTE N17:5/6 EOR
%   T4:18  ADS_B_BED_LT_ALM_TM  "TIMER Regen ADS B Wall Low Temp Alarm Delay" %
%   N17:5/6  LT_BED_ADS_B_ALARM  "ALARM ADS B Wall Low Temperature" %
%   B31:4/0  REGEN_RESUME  "COMMAND HMI Regen Resume" %
% Rung: 10 %
% ADS B Low Temp Bed Warning %
SOR EQU N17:0 N9:42 LEQ I:4.6 N7:45 XIC N13:5/2 BST XIO B38:0/0 NXB XIC B38:0/0 XIC B38:0/1 XIC B38:0/3 BND BST MOV N7:43 T4:19.PRE NXB XIC N7:4/9 TON T4:19 1.0 21600 0 BND EOR
%   N17:0  ADS_B_STATE  "STATE The current state of Adsorber B" %
%   N9:42  ADS_REGEN  "STATE ADS Regen" %
%   I:4.6  ADS_B_BED_TEMP  "TC8" %
%   N7:45  LT_ADS_BED_WRN_SP  "CONFIG ADS Wall Regen Heat Low Temperature Warning Setpoint" %
%   N13:5/2  REGEN_HEATER  "CONTROL Regen Operate the heater" %
%   B38:0/0  MAN_HTR_OVERRIDE %
%   B38:0/1  MAN_ADS_HTRS_ON %
%   B38:0/3  MAN_ADS_B_HTRS_ON %
%   N7:43  LT_ADS_BED_WRN_DLY  "CONFIG ADS Wall Regen heat Low Temperature Warning Delay" %
%   T4:19  ADS_B_BED_LT_WRN_TM  "TIMER Regen ADS B Wall Low Temp Warning Delay" %
%   N7:4/9  LT_ADS_BED_WRN_EN  "CONFIG ADS Wall Low Temperature Warning Enabled" %
% Rung: 11 %
SOR XIC T4:19/DN OTE N17:7/6 EOR
%   T4:19  ADS_B_BED_LT_WRN_TM  "TIMER Regen ADS B Wall Low Temp Warning Delay" %
%   N17:7/6  LT_BED_ADS_B_WARN  "WARNING ADS B Wall Low Temperature" %

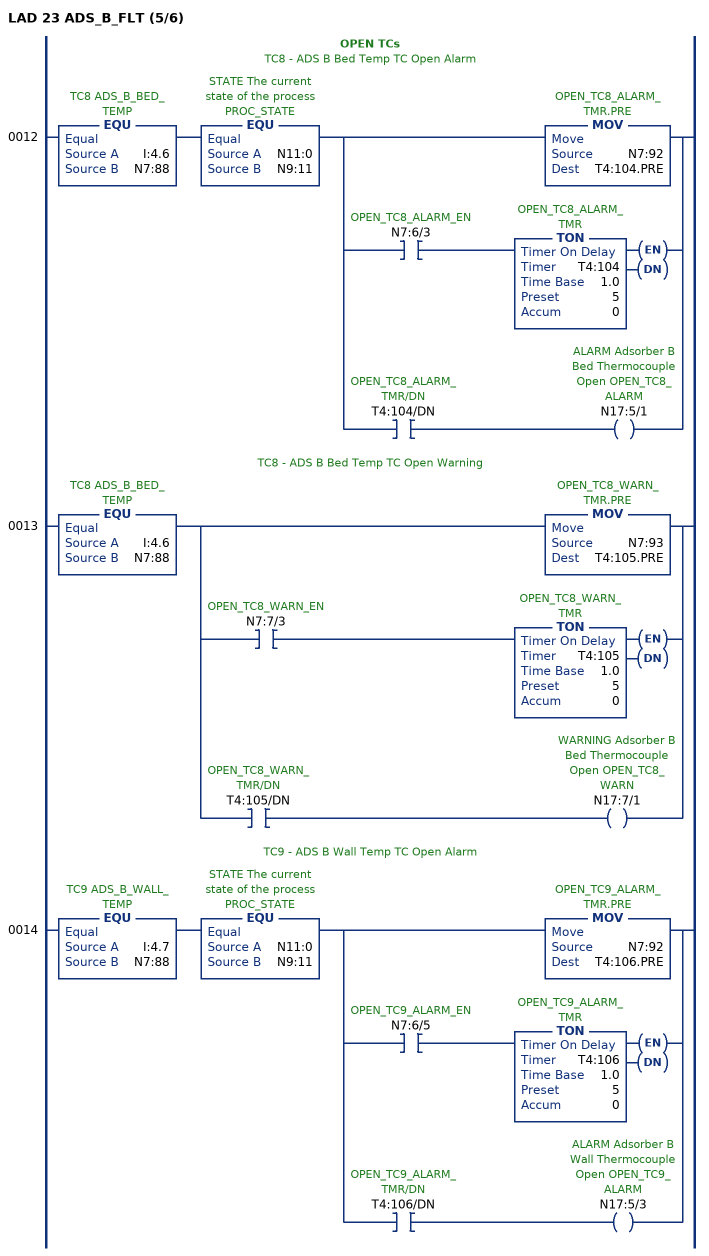
% Rung: 12 %
% TITLE: OPEN TCs %
% TC8 - ADS B Bed Temp TC Open Alarm %
SOR EQU I:4.6 N7:88 EQU N11:0 N9:11 BST MOV N7:92 T4:104.PRE NXB BST XIC N7:6/3 TON T4:104 1.0 5 0 NXB XIC T4:104/DN OTE N17:5/1 BND BND EOR
%   I:4.6  ADS_B_BED_TEMP  "TC8" %
%   N7:88  TC_OPEN_SP  "CONFIG The value read by an open TC input" %
%   N11:0  PROC_STATE  "STATE The current state of the process" %
%   N9:11  PROC_PURIFY_A  "STATE Process Purify A" %
%   N7:92  OPEN_TC_ALARM_DELAY %
%   T4:104  OPEN_TC8_ALARM_TMR %
%   N7:6/3  OPEN_TC8_ALARM_EN %
%   N17:5/1  OPEN_TC8_ALARM  "ALARM Adsorber B Bed Thermocouple Open" %
% Rung: 13 %
% TC8 - ADS B Bed Temp TC Open Warning %
SOR EQU I:4.6 N7:88 BST MOV N7:93 T4:105.PRE NXB BST XIC N7:7/3 TON T4:105 1.0 5 0 NXB XIC T4:105/DN OTE N17:7/1 BND BND EOR
%   I:4.6  ADS_B_BED_TEMP  "TC8" %
%   N7:88  TC_OPEN_SP  "CONFIG The value read by an open TC input" %
%   N7:93  OPEN_TC_WRN_DELAY %
%   T4:105  OPEN_TC8_WARN_TMR %
%   N7:7/3  OPEN_TC8_WARN_EN %
%   N17:7/1  OPEN_TC8_WARN  "WARNING Adsorber B Bed Thermocouple Open" %
% Rung: 14 %
% TC9 - ADS B Wall Temp TC Open Alarm %
SOR EQU I:4.7 N7:88 EQU N11:0 N9:11 BST MOV N7:92 T4:106.PRE NXB BST XIC N7:6/5 TON T4:106 1.0 5 0 NXB XIC T4:106/DN OTE N17:5/3 BND BND EOR
%   I:4.7  ADS_B_WALL_TEMP  "TC9" %
%   N7:88  TC_OPEN_SP  "CONFIG The value read by an open TC input" %
%   N11:0  PROC_STATE  "STATE The current state of the process" %
%   N9:11  PROC_PURIFY_A  "STATE Process Purify A" %
%   N7:92  OPEN_TC_ALARM_DELAY %
%   T4:106  OPEN_TC9_ALARM_TMR %
%   N7:6/5  OPEN_TC9_ALARM_EN %
%   N17:5/3  OPEN_TC9_ALARM  "ALARM Adsorber B Wall Thermocouple Open" %

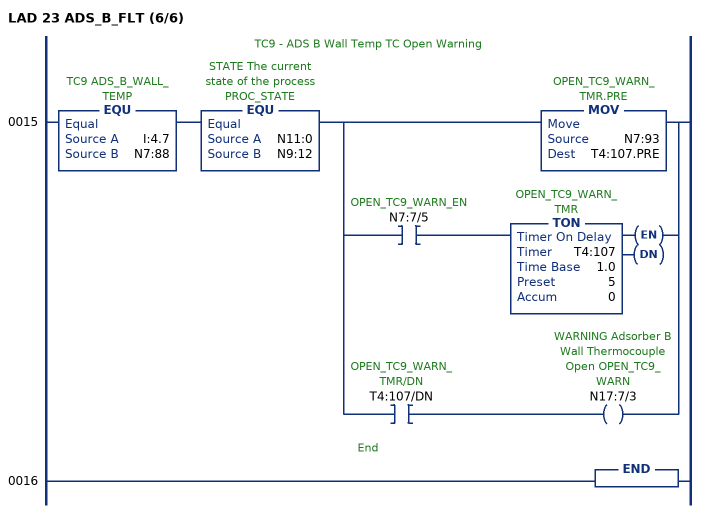
% Rung: 15 %
% TC9 - ADS B Wall Temp TC Open Warning %
SOR EQU I:4.7 N7:88 EQU N11:0 N9:12 BST MOV N7:93 T4:107.PRE NXB BST XIC N7:7/5 TON T4:107 1.0 5 0 NXB XIC T4:107/DN OTE N17:7/3 BND BND EOR
%   I:4.7  ADS_B_WALL_TEMP  "TC9" %
%   N7:88  TC_OPEN_SP  "CONFIG The value read by an open TC input" %
%   N11:0  PROC_STATE  "STATE The current state of the process" %
%   N9:12  PROC_PURIFY_B  "STATE Process Purify B" %
%   N7:93  OPEN_TC_WRN_DELAY %
%   T4:107  OPEN_TC9_WARN_TMR %
%   N7:7/5  OPEN_TC9_WARN_EN %
%   N17:7/3  OPEN_TC9_WARN  "WARNING Adsorber B Wall Thermocouple Open" %
% Rung: 16 %
% End %
SOR END EOR

LADDER 24 "PREHEATER"
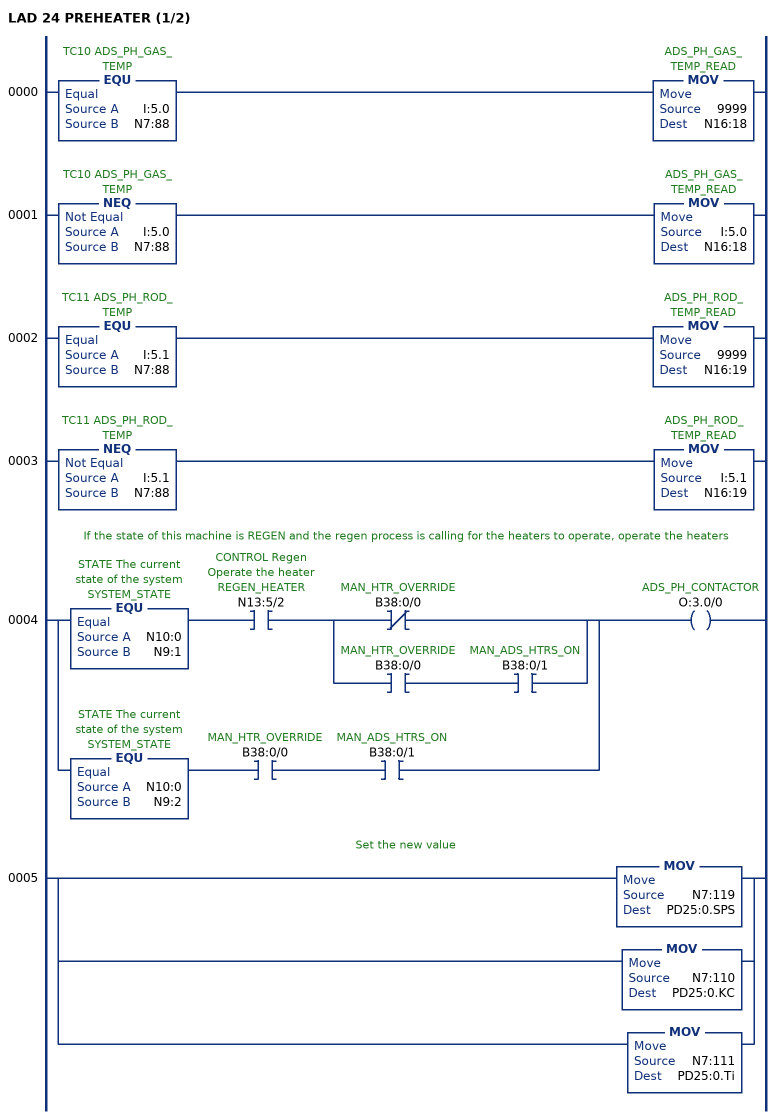
% Rung: 0 %
SOR EQU I:5.0 N7:88 MOV 9999 N16:18 EOR
%   I:5.0  ADS_PH_GAS_TEMP  "TC10" %
%   N7:88  TC_OPEN_SP  "CONFIG The value read by an open TC input" %
%   N16:18  ADS_PH_GAS_TEMP_READ %
% Rung: 1 %
SOR NEQ I:5.0 N7:88 MOV I:5.0 N16:18 EOR
%   I:5.0  ADS_PH_GAS_TEMP  "TC10" %
%   N7:88  TC_OPEN_SP  "CONFIG The value read by an open TC input" %
%   N16:18  ADS_PH_GAS_TEMP_READ %
% Rung: 2 %
SOR EQU I:5.1 N7:88 MOV 9999 N16:19 EOR
%   I:5.1  ADS_PH_ROD_TEMP  "TC11" %
%   N7:88  TC_OPEN_SP  "CONFIG The value read by an open TC input" %
%   N16:19  ADS_PH_ROD_TEMP_READ %
% Rung: 3 %
SOR NEQ I:5.1 N7:88 MOV I:5.1 N16:19 EOR
%   I:5.1  ADS_PH_ROD_TEMP  "TC11" %
%   N7:88  TC_OPEN_SP  "CONFIG The value read by an open TC input" %
%   N16:19  ADS_PH_ROD_TEMP_READ %
% Rung: 4 %
% If the state of this machine is REGEN and the regen process is calling for the heaters to operate, operate the heaters %
SOR BST EQU N10:0 N9:1 XIC N13:5/2 BST XIO B38:0/0 NXB XIC B38:0/0 XIC B38:0/1 BND NXB EQU N10:0 N9:2 XIC B38:0/0 XIC B38:0/1 BND OTE O:3.0/0 EOR
%   N10:0  SYSTEM_STATE  "STATE The current state of the system" %
%   N9:1  SYSTEM_PROCESS  "STATE System Process" %
%   N13:5/2  REGEN_HEATER  "CONTROL Regen Operate the heater" %
%   B38:0/0  MAN_HTR_OVERRIDE %
%   B38:0/1  MAN_ADS_HTRS_ON %
%   N9:2  SYSTEM_MANUAL  "STATE System Manual" %
%   O:3.0/0  ADS_PH_CONTACTOR %
% Rung: 5 %
% Set the new value %
SOR BST MOV N7:119 PD25:0.SPS NXB MOV N7:110 PD25:0.KC NXB MOV N7:111 PD25:0.Ti BND EOR
%   N7:119  PREHEATER_SP  "CONTROL Preheater PID Setpoint" %
%   N7:110  PREHEATER_P  "CONFIG Preheater Proportional Gain New" %
%   N7:111  PREHEATER_I  "CONFIG Preheater Integral Gain New" %

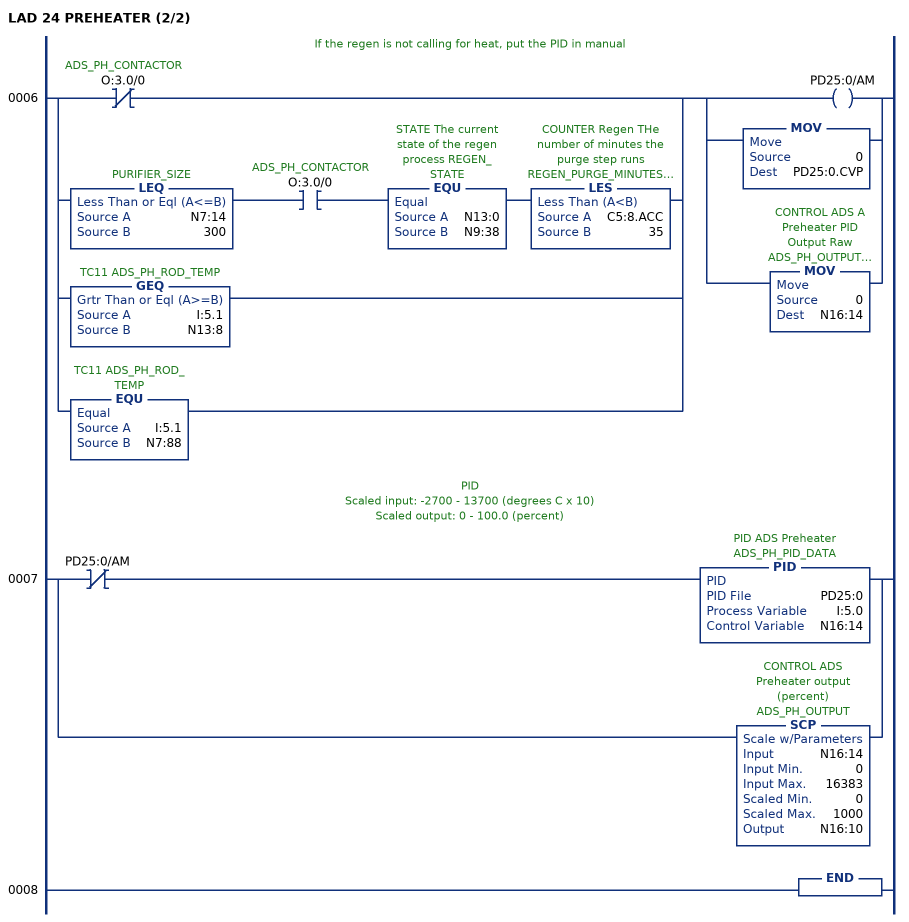
% Rung: 6 %
% If the regen is not calling for heat, put the PID in manual %
SOR BST XIO O:3.0/0 NXB LEQ N7:14 300 XIC O:3.0/0 EQU N13:0 N9:38 LES C5:8.ACC 35 NXB GEQ I:5.1 N13:8 NXB EQU I:5.1 N7:88 BND BST OTE PD25:0/AM NXB MOV 0 PD25:0.CVP NXB MOV 0 N16:14 BND EOR
%   O:3.0/0  ADS_PH_CONTACTOR %
%   N7:14  PURIFIER_SIZE %
%   N13:0  REGEN_STATE  "STATE The current state of the regen process" %
%   N9:38  REGEN_PURGE  "STATE Regen Hot Purge" %
%   C5:8  REGEN_PURGE_MINUTES  "COUNTER Regen THe number of minutes the purge step runs" %
%   I:5.1  ADS_PH_ROD_TEMP  "TC11" %
%   N13:8  PH_ROD_LIMIT %
%   N7:88  TC_OPEN_SP  "CONFIG The value read by an open TC input" %
%   N16:14  ADS_PH_OUTPUT_RAW  "CONTROL ADS A Preheater PID Output Raw" %
% Rung: 7 %
% PID
% Scaled input: -2700 - 13700 (degrees C x 10)
% Scaled output: 0 - 100.0 (percent) %
SOR BST XIO PD25:0/AM PID PD25:0 I:5.0 N16:14 NXB SCP N16:14 0 16383 0 1000 N16:10 BND EOR
%   PD25:0  ADS_PH_PID_DATA  "PID ADS Preheater" %
%   I:5.0  ADS_PH_GAS_TEMP  "TC10" %
%   N16:14  ADS_PH_OUTPUT_RAW  "CONTROL ADS A Preheater PID Output Raw" %
%   N16:10  ADS_PH_OUTPUT  "CONTROL ADS Preheater output (percent)" %
% Rung: 8 %
SOR END EOR

LADDER 25 "PH_FLT"
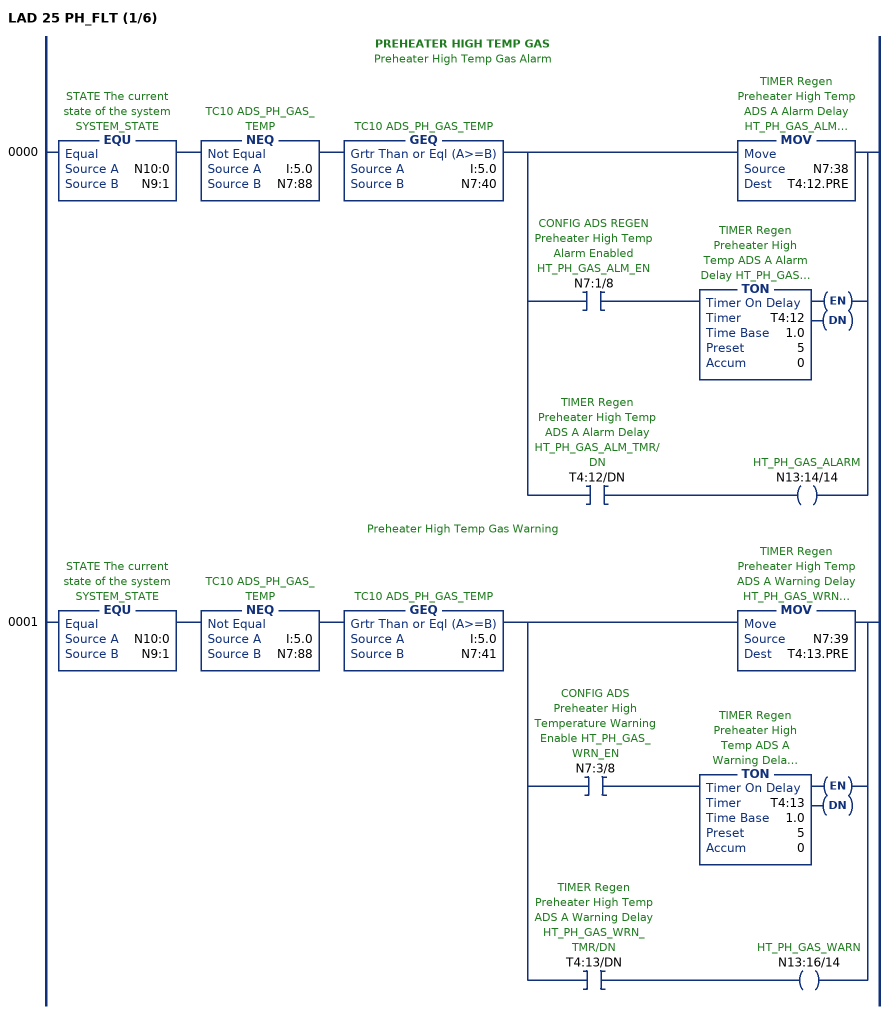
% Rung: 0 %
% TITLE: PREHEATER HIGH TEMP GAS %
% Preheater High Temp Gas Alarm %
SOR EQU N10:0 N9:1 NEQ I:5.0 N7:88 GEQ I:5.0 N7:40 BST MOV N7:38 T4:12.PRE NXB XIC N7:1/8 TON T4:12 1.0 5 0 NXB XIC T4:12/DN OTE N13:14/14 BND EOR
%   N10:0  SYSTEM_STATE  "STATE The current state of the system" %
%   N9:1  SYSTEM_PROCESS  "STATE System Process" %
%   I:5.0  ADS_PH_GAS_TEMP  "TC10" %
%   N7:88  TC_OPEN_SP  "CONFIG The value read by an open TC input" %
%   N7:40  HT_PH_GAS_ALM_SP  "CONFIG ADS Preheater High Temperature Alarm Temperature" %
%   N7:38  HT_PH_GAS_ALM_DLY  "CONFIG ADS Preheater High Temperature Alarm Delay" %
%   T4:12  HT_PH_GAS_ALM_TMR  "TIMER Regen Preheater High Temp ADS A Alarm Delay" %
%   N7:1/8  HT_PH_GAS_ALM_EN  "CONFIG ADS REGEN Preheater High Temp Alarm Enabled" %
%   N13:14/14  HT_PH_GAS_ALARM %
% Rung: 1 %
% Preheater High Temp Gas Warning %
SOR EQU N10:0 N9:1 NEQ I:5.0 N7:88 GEQ I:5.0 N7:41 BST MOV N7:39 T4:13.PRE NXB XIC N7:3/8 TON T4:13 1.0 5 0 NXB XIC T4:13/DN OTE N13:16/14 BND EOR
%   N10:0  SYSTEM_STATE  "STATE The current state of the system" %
%   N9:1  SYSTEM_PROCESS  "STATE System Process" %
%   I:5.0  ADS_PH_GAS_TEMP  "TC10" %
%   N7:88  TC_OPEN_SP  "CONFIG The value read by an open TC input" %
%   N7:41  HT_PH_GAS_WRN_SP  "CONFIG ADS Preheater High Temperature Warning Temperature" %
%   N7:39  HT_PH_GAS_WRN_DLY  "CONFIG ADS Preheater High Temperature Warning Delay" %
%   T4:13  HT_PH_GAS_WRN_TMR  "TIMER Regen Preheater High Temp ADS A Warning Delay" %
%   N7:3/8  HT_PH_GAS_WRN_EN  "CONFIG ADS Preheater High Temperature Warning Enable" %
%   N13:16/14  HT_PH_GAS_WARN %

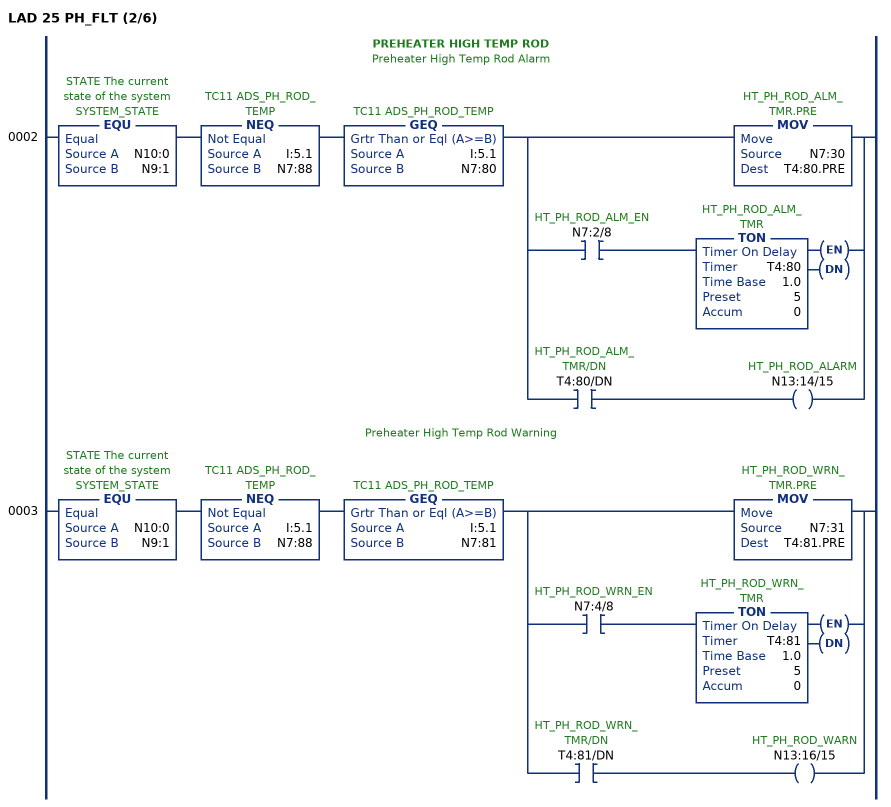
% Rung: 2 %
% TITLE: PREHEATER HIGH TEMP ROD %
% Preheater High Temp Rod Alarm %
SOR EQU N10:0 N9:1 NEQ I:5.1 N7:88 GEQ I:5.1 N7:80 BST MOV N7:30 T4:80.PRE NXB XIC N7:2/8 TON T4:80 1.0 5 0 NXB XIC T4:80/DN OTE N13:14/15 BND EOR
%   N10:0  SYSTEM_STATE  "STATE The current state of the system" %
%   N9:1  SYSTEM_PROCESS  "STATE System Process" %
%   I:5.1  ADS_PH_ROD_TEMP  "TC11" %
%   N7:88  TC_OPEN_SP  "CONFIG The value read by an open TC input" %
%   N7:80  HT_PH_ROD_ALM_SP %
%   N7:30  HT_PH_ROD_ALM_DLY %
%   T4:80  HT_PH_ROD_ALM_TMR %
%   N7:2/8  HT_PH_ROD_ALM_EN %
%   N13:14/15  HT_PH_ROD_ALARM %
% Rung: 3 %
% Preheater High Temp Rod Warning %
SOR EQU N10:0 N9:1 NEQ I:5.1 N7:88 GEQ I:5.1 N7:81 BST MOV N7:31 T4:81.PRE NXB XIC N7:4/8 TON T4:81 1.0 5 0 NXB XIC T4:81/DN OTE N13:16/15 BND EOR
%   N10:0  SYSTEM_STATE  "STATE The current state of the system" %
%   N9:1  SYSTEM_PROCESS  "STATE System Process" %
%   I:5.1  ADS_PH_ROD_TEMP  "TC11" %
%   N7:88  TC_OPEN_SP  "CONFIG The value read by an open TC input" %
%   N7:81  HT_PH_ROD_WRN_SP %
%   N7:31  HT_PH_ROD_WRN_DLY %
%   T4:81  HT_PH_ROD_WRN_TMR %
%   N7:4/8  HT_PH_ROD_WRN_EN %
%   N13:16/15  HT_PH_ROD_WARN %

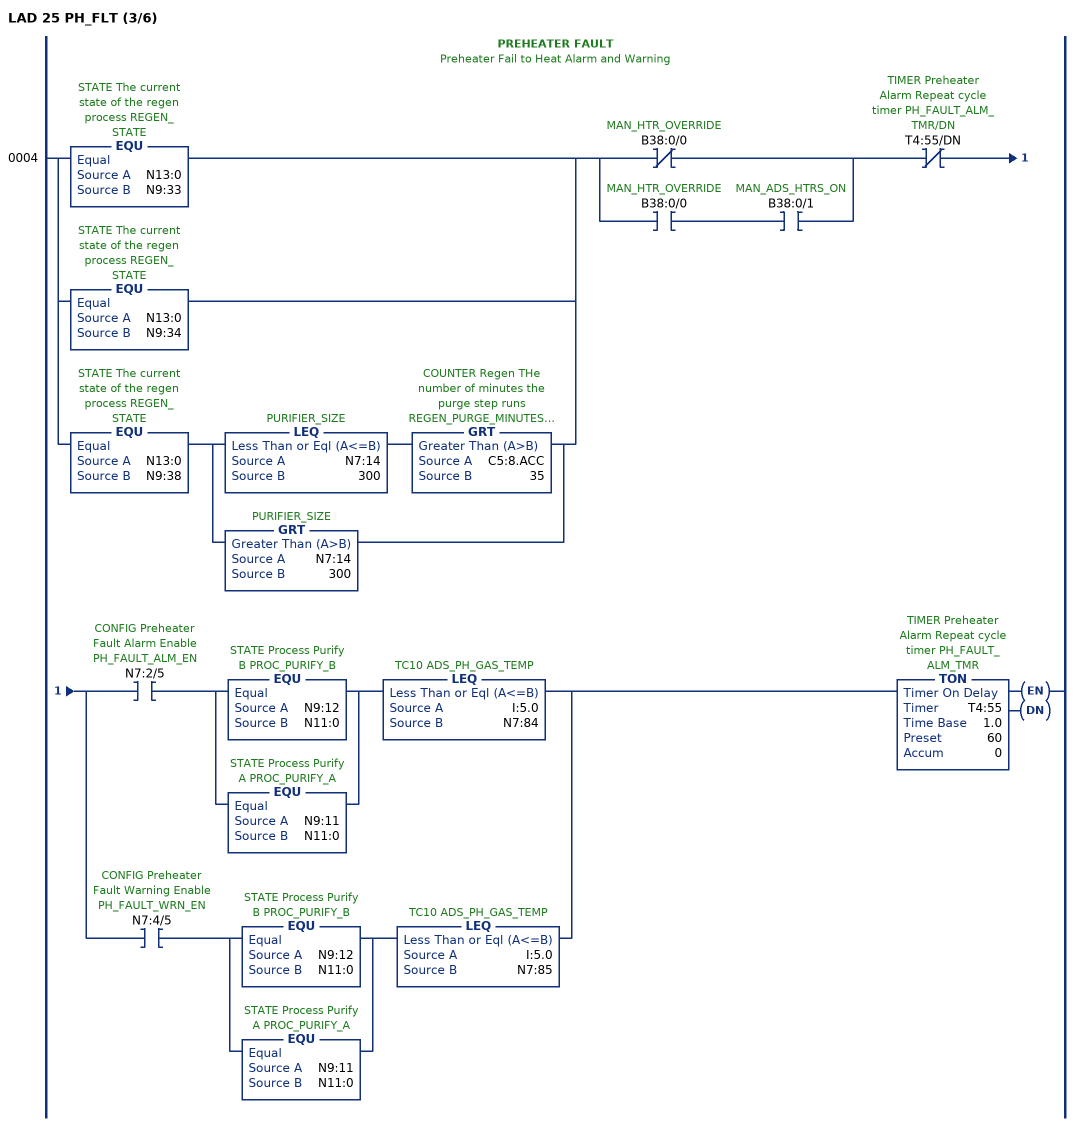
% Rung: 4 %
% TITLE: PREHEATER FAULT %
% Preheater Fail to Heat Alarm and Warning %
SOR BST EQU N13:0 N9:33 NXB EQU N13:0 N9:34 NXB EQU N13:0 N9:38 BST LEQ N7:14 300 GRT C5:8.ACC 35 NXB GRT N7:14 300 BND BND BST XIO B38:0/0 NXB XIC B38:0/0 XIC B38:0/1 BND XIO T4:55/DN BST XIC N7:2/5 BST EQU N9:12 N11:0 NXB EQU N9:11 N11:0 BND LEQ I:5.0 N7:84 NXB XIC N7:4/5 BST EQU N9:12 N11:0 NXB EQU N9:11 N11:0 BND LEQ I:5.0 N7:85 BND TON T4:55 1.0 60 0 EOR
%   N13:0  REGEN_STATE  "STATE The current state of the regen process" %
%   N9:33  REGEN_HEAT_BED  "STATE Regen Heat wall" %
%   N9:34  REGEN_H2_REDUCTION  "STATE Regen Running" %
%   N9:38  REGEN_PURGE  "STATE Regen Hot Purge" %
%   N7:14  PURIFIER_SIZE %
%   C5:8  REGEN_PURGE_MINUTES  "COUNTER Regen THe number of minutes the purge step runs" %
%   B38:0/0  MAN_HTR_OVERRIDE %
%   B38:0/1  MAN_ADS_HTRS_ON %
%   T4:55  PH_FAULT_ALM_TMR  "TIMER Preheater Alarm Repeat cycle timer" %
%   N7:2/5  PH_FAULT_ALM_EN  "CONFIG Preheater Fault Alarm Enable" %
%   N9:12  PROC_PURIFY_B  "STATE Process Purify B" %
%   N11:0  PROC_STATE  "STATE The current state of the process" %
%   N9:11  PROC_PURIFY_A  "STATE Process Purify A" %
%   I:5.0  ADS_PH_GAS_TEMP  "TC10" %
%   N7:84  PH_FAULT_ALARM_SP  "CONFIG Preheater Temperature Delta Alarm Setpoint" %
%   N7:4/5  PH_FAULT_WRN_EN  "CONFIG Preheater Fault Warning Enable" %
%   N7:85  PH_FAULT_WARN_SP %

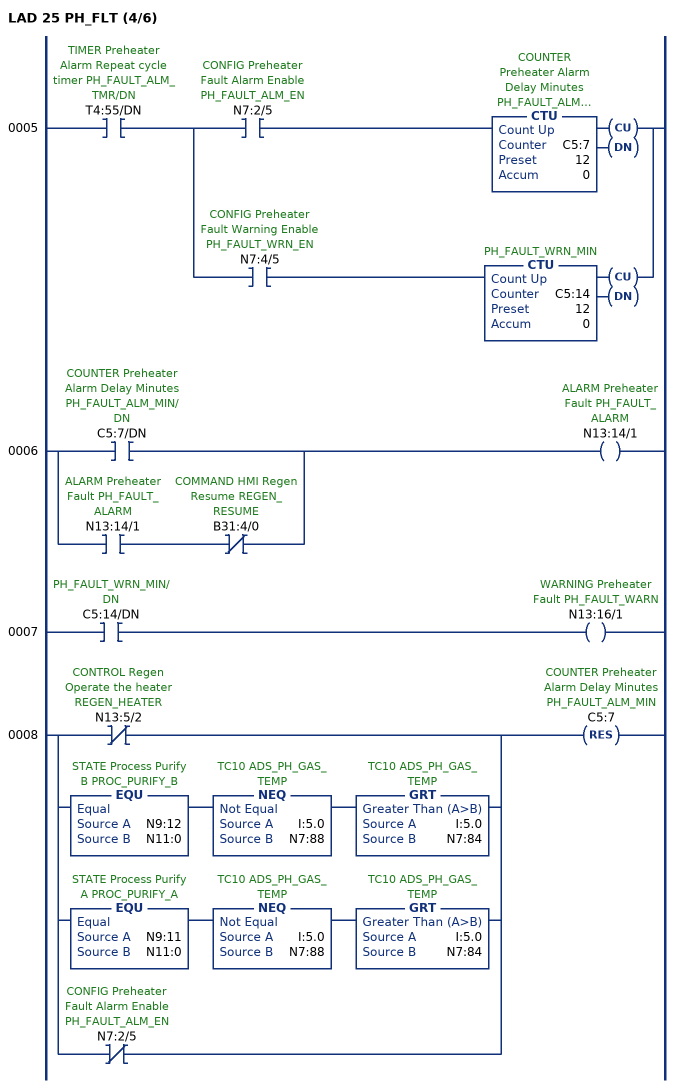
% Rung: 5 %
SOR XIC T4:55/DN BST XIC N7:2/5 CTU C5:7 12 0 NXB XIC N7:4/5 CTU C5:14 12 0 BND EOR
%   T4:55  PH_FAULT_ALM_TMR  "TIMER Preheater Alarm Repeat cycle timer" %
%   N7:2/5  PH_FAULT_ALM_EN  "CONFIG Preheater Fault Alarm Enable" %
%   C5:7  PH_FAULT_ALM_MIN  "COUNTER Preheater Alarm Delay Minutes" %
%   N7:4/5  PH_FAULT_WRN_EN  "CONFIG Preheater Fault Warning Enable" %
%   C5:14  PH_FAULT_WRN_MIN %
% Rung: 6 %
SOR BST XIC C5:7/DN NXB XIC N13:14/1 XIO B31:4/0 BND OTE N13:14/1 EOR
%   C5:7  PH_FAULT_ALM_MIN  "COUNTER Preheater Alarm Delay Minutes" %
%   N13:14/1  PH_FAULT_ALARM  "ALARM Preheater Fault" %
%   B31:4/0  REGEN_RESUME  "COMMAND HMI Regen Resume" %
% Rung: 7 %
SOR XIC C5:14/DN OTE N13:16/1 EOR
%   C5:14  PH_FAULT_WRN_MIN %
%   N13:16/1  PH_FAULT_WARN  "WARNING Preheater Fault" %
% Rung: 8 %
SOR BST XIO N13:5/2 NXB EQU N9:12 N11:0 NEQ I:5.0 N7:88 GRT I:5.0 N7:84 NXB EQU N9:11 N11:0 NEQ I:5.0 N7:88 GRT I:5.0 N7:84 NXB XIO N7:2/5 BND RES C5:7 EOR
%   N13:5/2  REGEN_HEATER  "CONTROL Regen Operate the heater" %
%   N9:12  PROC_PURIFY_B  "STATE Process Purify B" %
%   N11:0  PROC_STATE  "STATE The current state of the process" %
%   I:5.0  ADS_PH_GAS_TEMP  "TC10" %
%   N7:88  TC_OPEN_SP  "CONFIG The value read by an open TC input" %
%   N7:84  PH_FAULT_ALARM_SP  "CONFIG Preheater Temperature Delta Alarm Setpoint" %
%   N9:11  PROC_PURIFY_A  "STATE Process Purify A" %
%   N7:2/5  PH_FAULT_ALM_EN  "CONFIG Preheater Fault Alarm Enable" %
%   C5:7  PH_FAULT_ALM_MIN  "COUNTER Preheater Alarm Delay Minutes" %

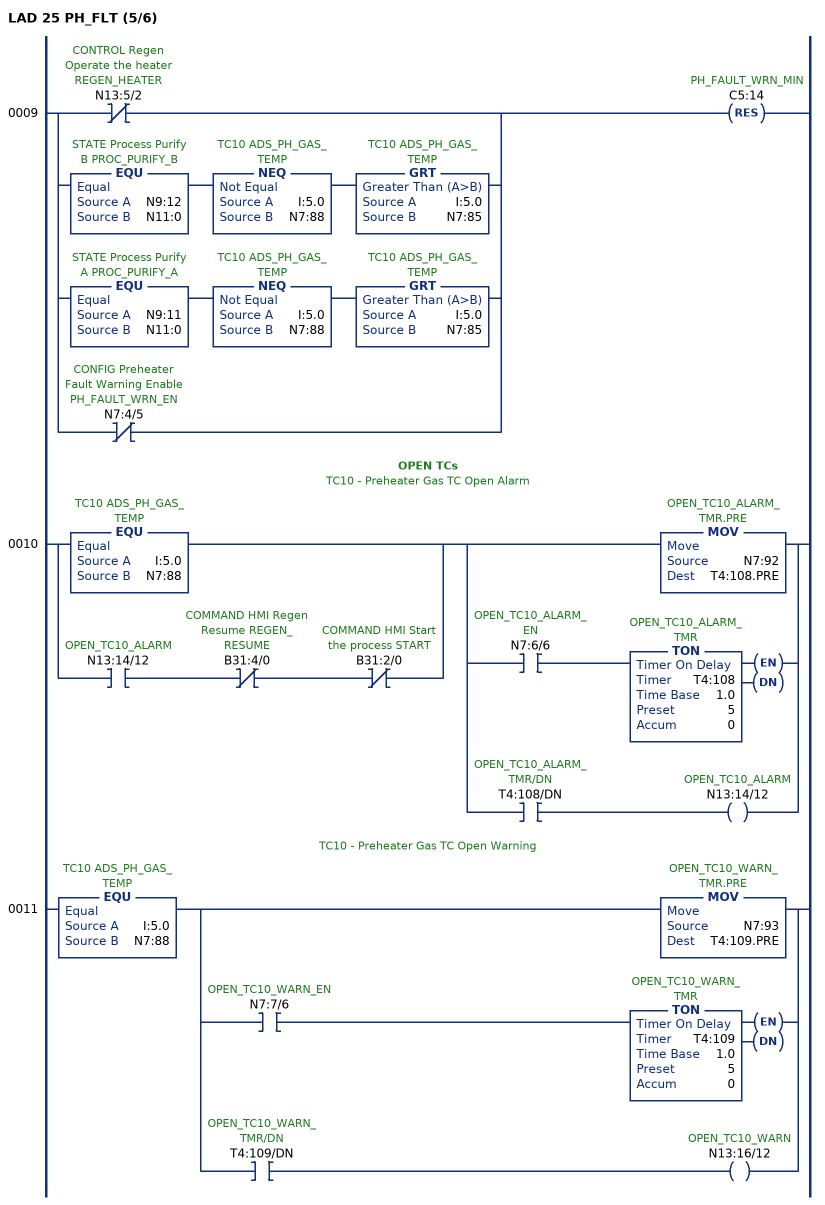
% Rung: 9 %
SOR BST XIO N13:5/2 NXB EQU N9:12 N11:0 NEQ I:5.0 N7:88 GRT I:5.0 N7:85 NXB EQU N9:11 N11:0 NEQ I:5.0 N7:88 GRT I:5.0 N7:85 NXB XIO N7:4/5 BND RES C5:14 EOR
%   N13:5/2  REGEN_HEATER  "CONTROL Regen Operate the heater" %
%   N9:12  PROC_PURIFY_B  "STATE Process Purify B" %
%   N11:0  PROC_STATE  "STATE The current state of the process" %
%   I:5.0  ADS_PH_GAS_TEMP  "TC10" %
%   N7:88  TC_OPEN_SP  "CONFIG The value read by an open TC input" %
%   N7:85  PH_FAULT_WARN_SP %
%   N9:11  PROC_PURIFY_A  "STATE Process Purify A" %
%   N7:4/5  PH_FAULT_WRN_EN  "CONFIG Preheater Fault Warning Enable" %
%   C5:14  PH_FAULT_WRN_MIN %
% Rung: 10 %
% TITLE: OPEN TCs %
% TC10 - Preheater Gas TC Open Alarm %
SOR BST EQU I:5.0 N7:88 NXB XIC N13:14/12 XIO B31:4/0 XIO B31:2/0 BND BST MOV N7:92 T4:108.PRE NXB BST XIC N7:6/6 TON T4:108 1.0 5 0 NXB XIC T4:108/DN OTE N13:14/12 BND BND EOR
%   I:5.0  ADS_PH_GAS_TEMP  "TC10" %
%   N7:88  TC_OPEN_SP  "CONFIG The value read by an open TC input" %
%   N13:14/12  OPEN_TC10_ALARM %
%   B31:4/0  REGEN_RESUME  "COMMAND HMI Regen Resume" %
%   B31:2/0  START  "COMMAND HMI Start the process" %
%   N7:92  OPEN_TC_ALARM_DELAY %
%   T4:108  OPEN_TC10_ALARM_TMR %
%   N7:6/6  OPEN_TC10_ALARM_EN %
% Rung: 11 %
% TC10 - Preheater Gas TC Open Warning %
SOR EQU I:5.0 N7:88 BST MOV N7:93 T4:109.PRE NXB BST XIC N7:7/6 TON T4:109 1.0 5 0 NXB XIC T4:109/DN OTE N13:16/12 BND BND EOR
%   I:5.0  ADS_PH_GAS_TEMP  "TC10" %
%   N7:88  TC_OPEN_SP  "CONFIG The value read by an open TC input" %
%   N7:93  OPEN_TC_WRN_DELAY %
%   T4:109  OPEN_TC10_WARN_TMR %
%   N7:7/6  OPEN_TC10_WARN_EN %
%   N13:16/12  OPEN_TC10_WARN %

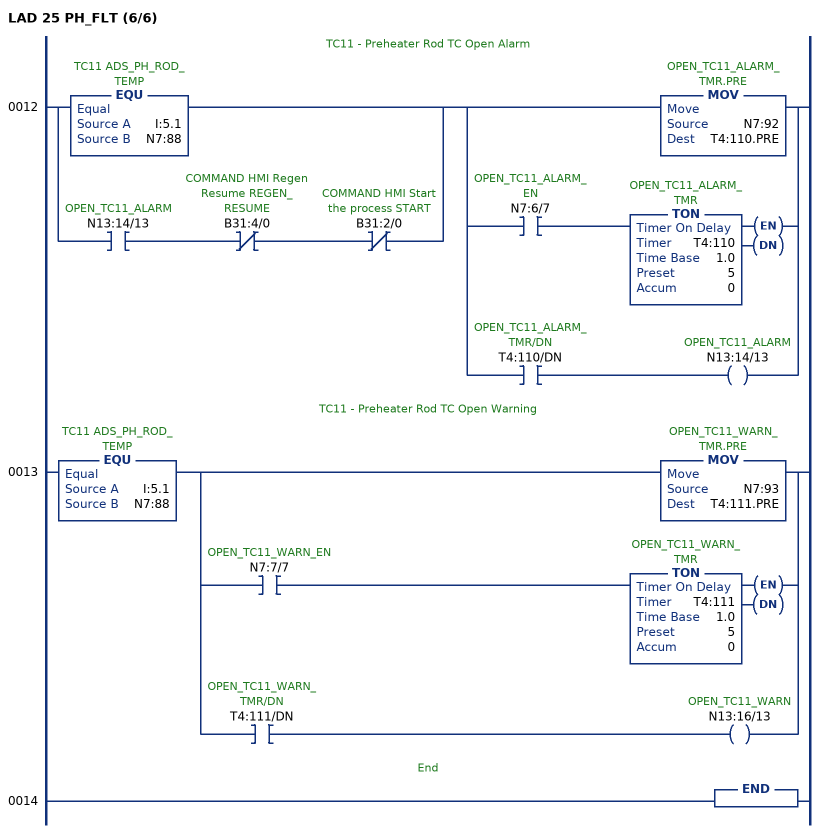
% Rung: 12 %
% TC11 - Preheater Rod TC Open Alarm %
SOR BST EQU I:5.1 N7:88 NXB XIC N13:14/13 XIO B31:4/0 XIO B31:2/0 BND BST MOV N7:92 T4:110.PRE NXB BST XIC N7:6/7 TON T4:110 1.0 5 0 NXB XIC T4:110/DN OTE N13:14/13 BND BND EOR
%   I:5.1  ADS_PH_ROD_TEMP  "TC11" %
%   N7:88  TC_OPEN_SP  "CONFIG The value read by an open TC input" %
%   N13:14/13  OPEN_TC11_ALARM %
%   B31:4/0  REGEN_RESUME  "COMMAND HMI Regen Resume" %
%   B31:2/0  START  "COMMAND HMI Start the process" %
%   N7:92  OPEN_TC_ALARM_DELAY %
%   T4:110  OPEN_TC11_ALARM_TMR %
%   N7:6/7  OPEN_TC11_ALARM_EN %
% Rung: 13 %
% TC11 - Preheater Rod TC Open Warning %
SOR EQU I:5.1 N7:88 BST MOV N7:93 T4:111.PRE NXB BST XIC N7:7/7 TON T4:111 1.0 5 0 NXB XIC T4:111/DN OTE N13:16/13 BND BND EOR
%   I:5.1  ADS_PH_ROD_TEMP  "TC11" %
%   N7:88  TC_OPEN_SP  "CONFIG The value read by an open TC input" %
%   N7:93  OPEN_TC_WRN_DELAY %
%   T4:111  OPEN_TC11_WARN_TMR %
%   N7:7/7  OPEN_TC11_WARN_EN %
%   N13:16/13  OPEN_TC11_WARN %
% Rung: 14 %
% End %
SOR END EOR

LADDER 49 "MODBUS"
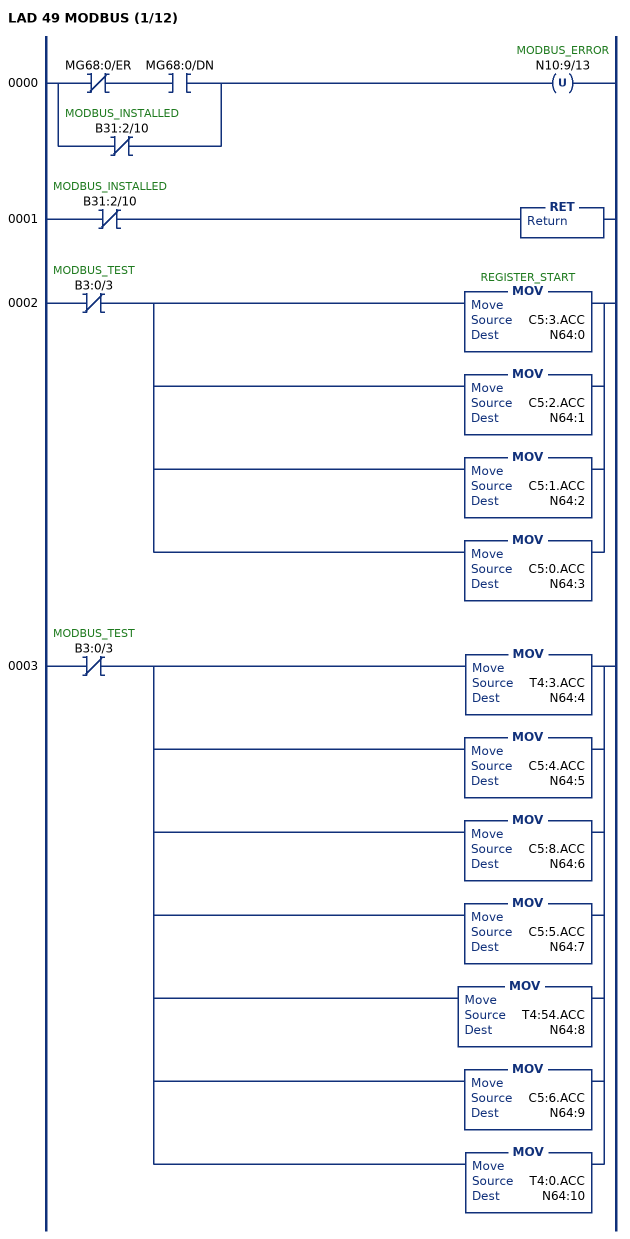
% Rung: 0 %
SOR BST XIO MG68:0/ER XIC MG68:0/DN NXB XIO B31:2/10 BND OTU N10:9/13 EOR
%   B31:2/10  MODBUS_INSTALLED %
%   N10:9/13  MODBUS_ERROR %
% Rung: 1 %
SOR XIO B31:2/10 RET EOR
%   B31:2/10  MODBUS_INSTALLED %
% Rung: 2 %
SOR XIO B3:0/3 BST MOV C5:3.ACC N64:0 NXB MOV C5:2.ACC N64:1 NXB MOV C5:1.ACC N64:2 NXB MOV C5:0.ACC N64:3 BND EOR
%   B3:0/3  MODBUS_TEST %
%   C5:3  PURIFY_ACTIVE_TTL_DY  "COUNTER The number of total elapsed purification days for the process equipment" %
%   N64:0  REGISTER_START %
%   C5:2  PURIFY_ACTIVE_TTL_HR  "COUNTER The number of total elapsed purification hours for the process equipment" %
%   C5:1  PURIFY_ACTIVE_MINUTE  "COUNTER The number of elapsed purification minutes for the current ADS (60 min)" %
%   C5:0  PURIFY_ACTIVE_HOURS  "COUNTER The number of elapsed purification hours for the current ADS" %
% Rung: 3 %
SOR XIO B3:0/3 BST MOV T4:3.ACC N64:4 NXB MOV C5:4.ACC N64:5 NXB MOV C5:8.ACC N64:6 NXB MOV C5:5.ACC N64:7 NXB MOV T4:54.ACC N64:8 NXB MOV C5:6.ACC N64:9 NXB MOV T4:0.ACC N64:10 BND EOR
%   B3:0/3  MODBUS_TEST %
%   T4:3  REGEN_VENT_TIMER  "TIMER Regen Vent (seconds)" %
%   C5:4  REGEN_REDUC_MINUTE  "COUNTER Regen The number of minutes which the regen reduc runs" %
%   C5:8  REGEN_PURGE_MINUTES  "COUNTER Regen THe number of minutes the purge step runs" %
%   C5:5  REGEN_COOL_MINUTE  "COUNTER Regen the number of minutes for which the bed has cooled" %
%   T4:54  REGEN_VENT_2_TMR %
%   C5:6  REGEN_EQUALIZE_MIN %
%   T4:0  PURIFY_OVERLAP_TIMER  "TIMER Purify Overlap" %

